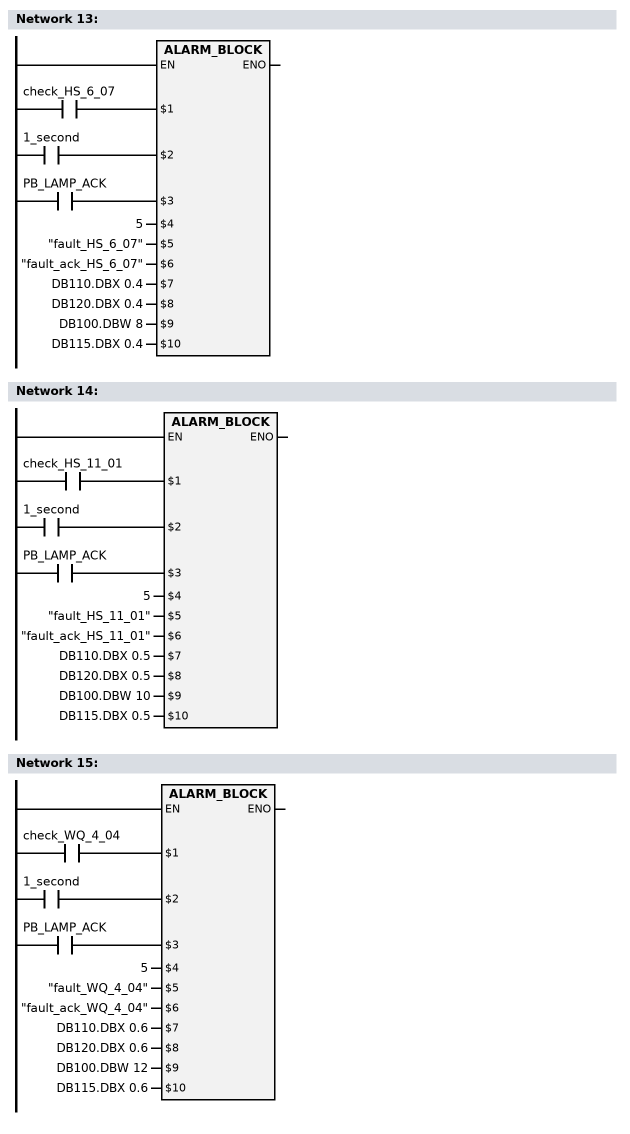
[picture p24: ALARM_HANDLING_STARCH networks 13-15]
NETWORK
TITLE =
      A     "check_HS_6_07";
      =     L 0.0;
      BLD   103;
      A     "1_second";
      =     L 0.1;
      BLD   103;
      A     "PB_LAMP_ACK";
      =     L 0.2;
      BLD   103;
      CALL  "ALARM_BLOCK" (
           $1                       := L 0.0,
           $2                       := L 0.1,
           $3                       := L 0.2,
           $4                       := 5,
           $5                       := "fault_HS_6_07",
           $6                       := "fault_ack_HS_6_07",
           $7                       := DB110.DBX 0.4,
           $8                       := DB120.DBX 0.4,
           $9                       := DB100.DBW 8,
           $10                      := DB115.DBX 0.4);
      NOP   0;
NETWORK
TITLE =
      A     "check_HS_11_01";
      =     L 0.0;
      BLD   103;
      A     "1_second";
      =     L 0.1;
      BLD   103;
      A     "PB_LAMP_ACK";
      =     L 0.2;
      BLD   103;
      CALL  "ALARM_BLOCK" (
           $1                       := L 0.0,
           $2                       := L 0.1,
           $3                       := L 0.2,
           $4                       := 5,
           $5                       := "fault_HS_11_01",
           $6                       := "fault_ack_HS_11_01",
           $7                       := DB110.DBX 0.5,
           $8                       := DB120.DBX 0.5,
           $9                       := DB100.DBW 10,
           $10                      := DB115.DBX 0.5);
      NOP   0;
NETWORK
TITLE =
      A     "check_WQ_4_04";
      =     L 0.0;
      BLD   103;
      A     "1_second";
      =     L 0.1;
      BLD   103;
      A     "PB_LAMP_ACK";
      =     L 0.2;
      BLD   103;
      CALL  "ALARM_BLOCK" (
           $1                       := L 0.0,
           $2                       := L 0.1,
           $3                       := L 0.2,
           $4                       := 5,
           $5                       := "fault_WQ_4_04",
           $6                       := "fault_ack_WQ_4_04",
           $7                       := DB110.DBX 0.6,
           $8                       := DB120.DBX 0.6,
           $9                       := DB100.DBW 12,
           $10                      := DB115.DBX 0.6);
      NOP   0;
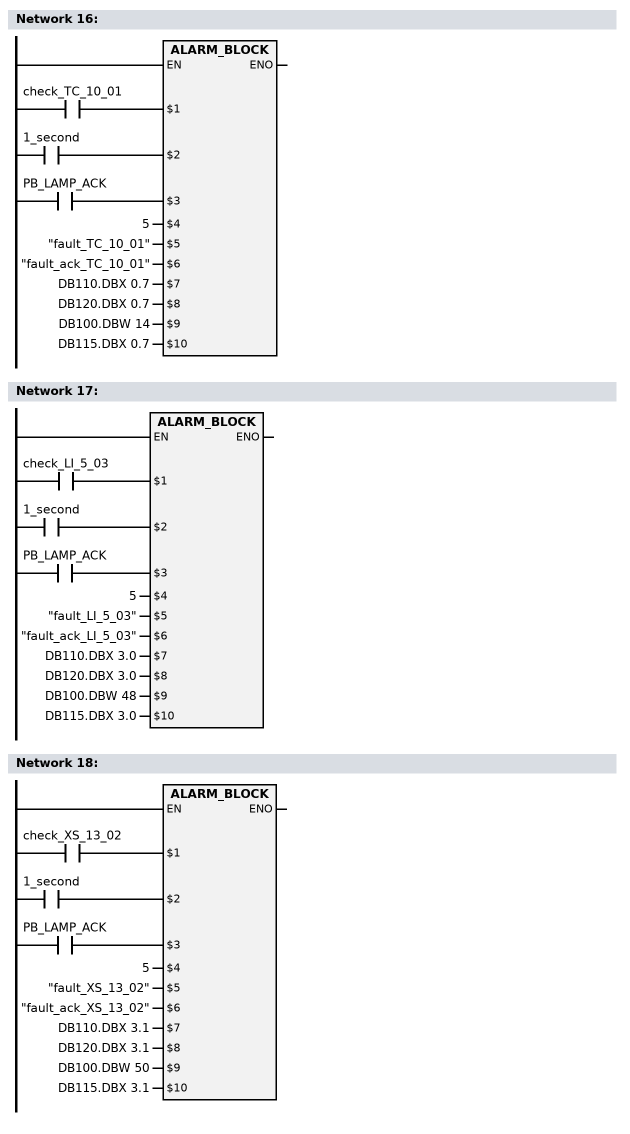
NETWORK
TITLE =
      A     "check_TC_10_01";
      =     L 0.0;
      BLD   103;
      A     "1_second";
      =     L 0.1;
      BLD   103;
      A     "PB_LAMP_ACK";
      =     L 0.2;
      BLD   103;
      CALL  "ALARM_BLOCK" (
           $1                       := L 0.0,
           $2                       := L 0.1,
           $3                       := L 0.2,
           $4                       := 5,
           $5                       := "fault_TC_10_01",
           $6                       := "fault_ack_TC_10_01",
           $7                       := DB110.DBX 0.7,
           $8                       := DB120.DBX 0.7,
           $9                       := DB100.DBW 14,
           $10                      := DB115.DBX 0.7);
      NOP   0;
NETWORK
TITLE =
      A     "check_LI_5_03";
      =     L 0.0;
      BLD   103;
      A     "1_second";
      =     L 0.1;
      BLD   103;
      A     "PB_LAMP_ACK";
      =     L 0.2;
      BLD   103;
      CALL  "ALARM_BLOCK" (
           $1                       := L 0.0,
           $2                       := L 0.1,
           $3                       := L 0.2,
           $4                       := 5,
           $5                       := "fault_LI_5_03",
           $6                       := "fault_ack_LI_5_03",
           $7                       := DB110.DBX 3.0,
           $8                       := DB120.DBX 3.0,
           $9                       := DB100.DBW 48,
           $10                      := DB115.DBX 3.0);
      NOP   0;
NETWORK
TITLE =
      A     "check_XS_13_02";
      =     L 0.0;
      BLD   103;
      A     "1_second";
      =     L 0.1;
      BLD   103;
      A     "PB_LAMP_ACK";
      =     L 0.2;
      BLD   103;
      CALL  "ALARM_BLOCK" (
           $1                       := L 0.0,
           $2                       := L 0.1,
           $3                       := L 0.2,
           $4                       := 5,
           $5                       := "fault_XS_13_02",
           $6                       := "fault_ack_XS_13_02",
           $7                       := DB110.DBX 3.1,
           $8                       := DB120.DBX 3.1,
           $9                       := DB100.DBW 50,
           $10                      := DB115.DBX 3.1);
      NOP   0;
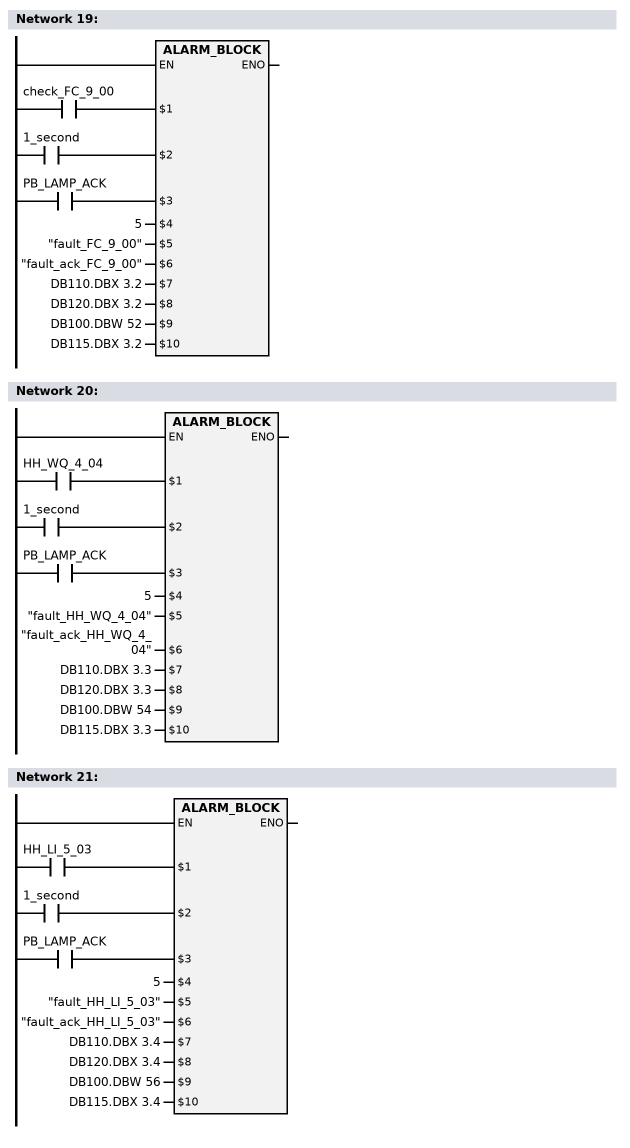
NETWORK
TITLE =
      A     "check_FC_9_00";
      =     L 0.0;
      BLD   103;
      A     "1_second";
      =     L 0.1;
      BLD   103;
      A     "PB_LAMP_ACK";
      =     L 0.2;
      BLD   103;
      CALL  "ALARM_BLOCK" (
           $1                       := L 0.0,
           $2                       := L 0.1,
           $3                       := L 0.2,
           $4                       := 5,
           $5                       := "fault_FC_9_00",
           $6                       := "fault_ack_FC_9_00",
           $7                       := DB110.DBX 3.2,
           $8                       := DB120.DBX 3.2,
           $9                       := DB100.DBW 52,
           $10                      := DB115.DBX 3.2);
      NOP   0;
NETWORK
TITLE =
      A     "HH_WQ_4_04";
      =     L 0.0;
      BLD   103;
      A     "1_second";
      =     L 0.1;
      BLD   103;
      A     "PB_LAMP_ACK";
      =     L 0.2;
      BLD   103;
      CALL  "ALARM_BLOCK" (
           $1                       := L 0.0,
           $2                       := L 0.1,
           $3                       := L 0.2,
           $4                       := 5,
           $5                       := "fault_HH_WQ_4_04",
           $6                       := "fault_ack_HH_WQ_4_04",
           $7                       := DB110.DBX 3.3,
           $8                       := DB120.DBX 3.3,
           $9                       := DB100.DBW 54,
           $10                      := DB115.DBX 3.3);
      NOP   0;
NETWORK
TITLE =
      A     "HH_LI_5_03";
      =     L 0.0;
      BLD   103;
      A     "1_second";
      =     L 0.1;
      BLD   103;
      A     "PB_LAMP_ACK";
      =     L 0.2;
      BLD   103;
      CALL  "ALARM_BLOCK" (
           $1                       := L 0.0,
           $2                       := L 0.1,
           $3                       := L 0.2,
           $4                       := 5,
           $5                       := "fault_HH_LI_5_03",
           $6                       := "fault_ack_HH_LI_5_03",
           $7                       := DB110.DBX 3.4,
           $8                       := DB120.DBX 3.4,
           $9                       := DB100.DBW 56,
           $10                      := DB115.DBX 3.4);
      NOP   0;
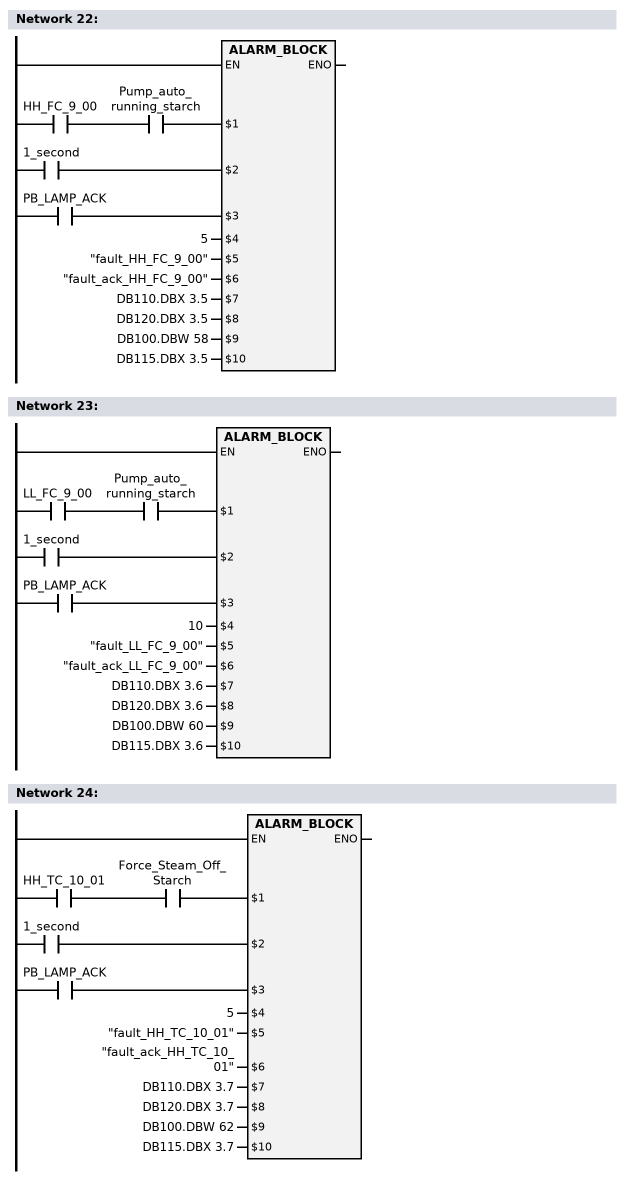
NETWORK
TITLE =
      A     "HH_FC_9_00";
      A     "Pump_auto_running_starch";
      =     L 0.0;
      BLD   103;
      A     "1_second";
      =     L 0.1;
      BLD   103;
      A     "PB_LAMP_ACK";
      =     L 0.2;
      BLD   103;
      CALL  "ALARM_BLOCK" (
           $1                       := L 0.0,
           $2                       := L 0.1,
           $3                       := L 0.2,
           $4                       := 5,
           $5                       := "fault_HH_FC_9_00",
           $6                       := "fault_ack_HH_FC_9_00",
           $7                       := DB110.DBX 3.5,
           $8                       := DB120.DBX 3.5,
           $9                       := DB100.DBW 58,
           $10                      := DB115.DBX 3.5);
      NOP   0;
NETWORK
TITLE =
      A     "LL_FC_9_00";
      A     "Pump_auto_running_starch";
      =     L 0.0;
      BLD   103;
      A     "1_second";
      =     L 0.1;
      BLD   103;
      A     "PB_LAMP_ACK";
      =     L 0.2;
      BLD   103;
      CALL  "ALARM_BLOCK" (
           $1                       := L 0.0,
           $2                       := L 0.1,
           $3                       := L 0.2,
           $4                       := 10,
           $5                       := "fault_LL_FC_9_00",
           $6                       := "fault_ack_LL_FC_9_00",
           $7                       := DB110.DBX 3.6,
           $8                       := DB120.DBX 3.6,
           $9                       := DB100.DBW 60,
           $10                      := DB115.DBX 3.6);
      NOP   0;
NETWORK
TITLE =
      A     "HH_TC_10_01";
      A     "Force_Steam_Off_Starch";
      =     L 0.0;
      BLD   103;
      A     "1_second";
      =     L 0.1;
      BLD   103;
      A     "PB_LAMP_ACK";
      =     L 0.2;
      BLD   103;
      CALL  "ALARM_BLOCK" (
           $1                       := L 0.0,
           $2                       := L 0.1,
           $3                       := L 0.2,
           $4                       := 5,
           $5                       := "fault_HH_TC_10_01",
           $6                       := "fault_ack_HH_TC_10_01",
           $7                       := DB110.DBX 3.7,
           $8                       := DB120.DBX 3.7,
           $9                       := DB100.DBW 62,
           $10                      := DB115.DBX 3.7);
      NOP   0;
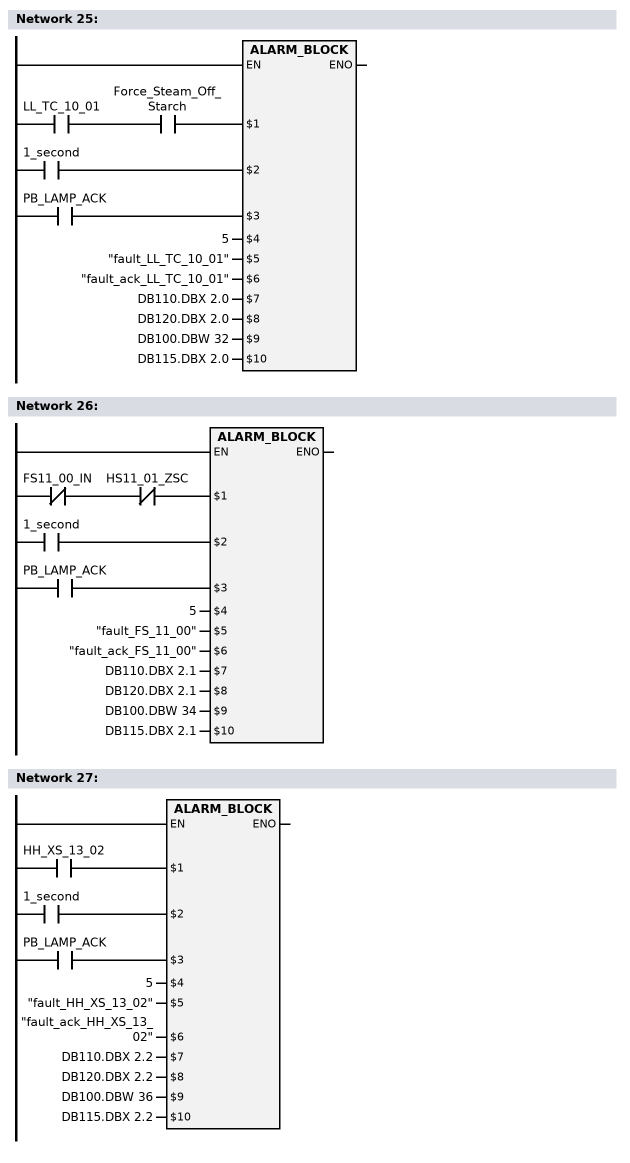
NETWORK
TITLE =
      A     "LL_TC_10_01";
      A     "Force_Steam_Off_Starch";
      =     L 0.0;
      BLD   103;
      A     "1_second";
      =     L 0.1;
      BLD   103;
      A     "PB_LAMP_ACK";
      =     L 0.2;
      BLD   103;
      CALL  "ALARM_BLOCK" (
           $1                       := L 0.0,
           $2                       := L 0.1,
           $3                       := L 0.2,
           $4                       := 5,
           $5                       := "fault_LL_TC_10_01",
           $6                       := "fault_ack_LL_TC_10_01",
           $7                       := DB110.DBX 2.0,
           $8                       := DB120.DBX 2.0,
           $9                       := DB100.DBW 32,
           $10                      := DB115.DBX 2.0);
      NOP   0;
NETWORK
TITLE =
      AN    "FS11_00_IN";
      AN    "HS11_01_ZSC";
      =     L 0.0;
      BLD   103;
      A     "1_second";
      =     L 0.1;
      BLD   103;
      A     "PB_LAMP_ACK";
      =     L 0.2;
      BLD   103;
      CALL  "ALARM_BLOCK" (
           $1                       := L 0.0,
           $2                       := L 0.1,
           $3                       := L 0.2,
           $4                       := 5,
           $5                       := "fault_FS_11_00",
           $6                       := "fault_ack_FS_11_00",
           $7                       := DB110.DBX 2.1,
           $8                       := DB120.DBX 2.1,
           $9                       := DB100.DBW 34,
           $10                      := DB115.DBX 2.1);
      NOP   0;
NETWORK
TITLE =
      A     "HH_XS_13_02";
      =     L 0.0;
      BLD   103;
      A     "1_second";
      =     L 0.1;
      BLD   103;
      A     "PB_LAMP_ACK";
      =     L 0.2;
      BLD   103;
      CALL  "ALARM_BLOCK" (
           $1                       := L 0.0,
           $2                       := L 0.1,
           $3                       := L 0.2,
           $4                       := 5,
           $5                       := "fault_HH_XS_13_02",
           $6                       := "fault_ack_HH_XS_13_02",
           $7                       := DB110.DBX 2.2,
           $8                       := DB120.DBX 2.2,
           $9                       := DB100.DBW 36,
           $10                      := DB115.DBX 2.2);
      NOP   0;
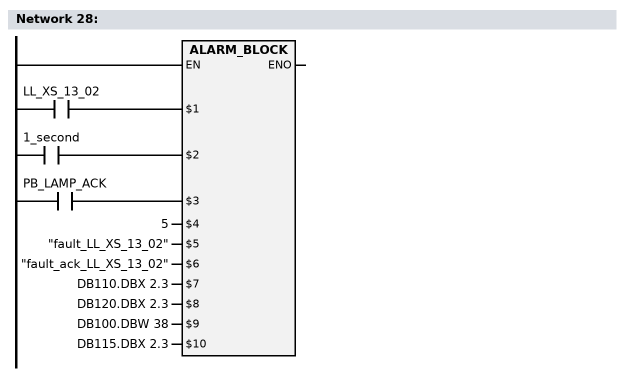
NETWORK
TITLE =
      A     "LL_XS_13_02";
      =     L 0.0;
      BLD   103;
      A     "1_second";
      =     L 0.1;
      BLD   103;
      A     "PB_LAMP_ACK";
      =     L 0.2;
      BLD   103;
      CALL  "ALARM_BLOCK" (
           $1                       := L 0.0,
           $2                       := L 0.1,
           $3                       := L 0.2,
           $4                       := 5,
           $5                       := "fault_LL_XS_13_02",
           $6                       := "fault_ack_LL_XS_13_02",
           $7                       := DB110.DBX 2.3,
           $8                       := DB120.DBX 2.3,
           $9                       := DB100.DBW 38,
           $10                      := DB115.DBX 2.3);
      NOP   0;
END_FUNCTION_BLOCK

FUNCTION_BLOCK "ALARM_HANDLING_CaCO3"	// FB 32
AUTHOR : GAW-LK
FAMILY : ALARM
NAME : ALARMS
VERSION : 0.1
BEGIN
// (block stored without names or comments; labels and parameter names are numbered)
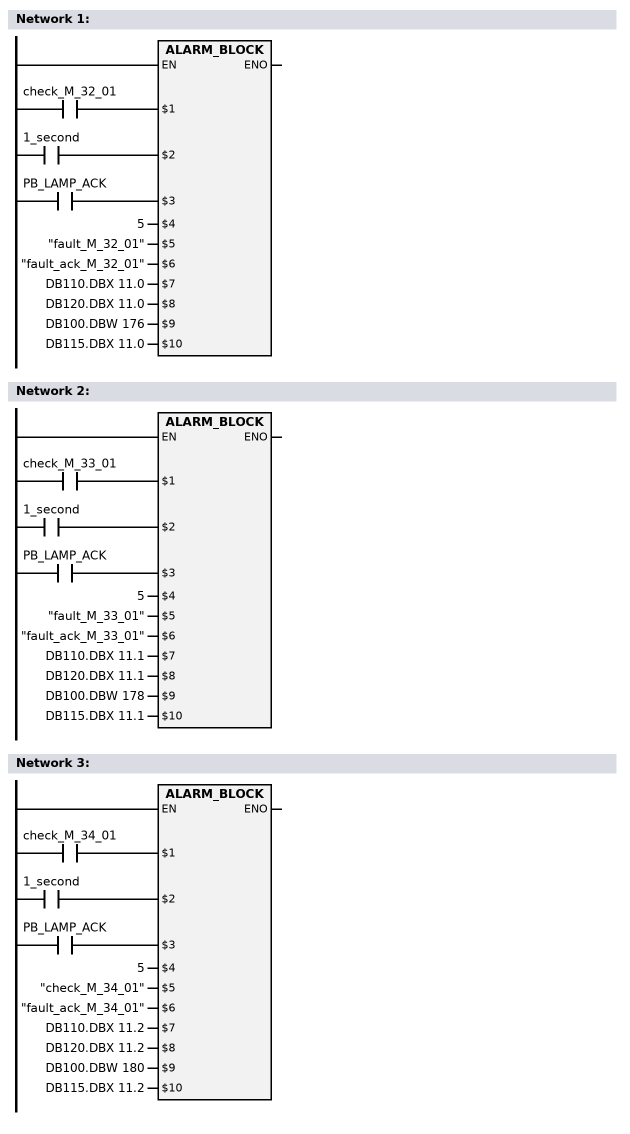
NETWORK
TITLE =
      A     "check_M_32_01";
      =     L 0.0;
      BLD   103;
      A     "1_second";
      =     L 0.1;
      BLD   103;
      A     "PB_LAMP_ACK";
      =     L 0.2;
      BLD   103;
      CALL  "ALARM_BLOCK" (
           $1                       := L 0.0,
           $2                       := L 0.1,
           $3                       := L 0.2,
           $4                       := 5,
           $5                       := "fault_M_32_01",
           $6                       := "fault_ack_M_32_01",
           $7                       := DB110.DBX 11.0,
           $8                       := DB120.DBX 11.0,
           $9                       := DB100.DBW 176,
           $10                      := DB115.DBX 11.0);
      NOP   0;
NETWORK
TITLE =
      A     "check_M_33_01";
      =     L 0.0;
      BLD   103;
      A     "1_second";
      =     L 0.1;
      BLD   103;
      A     "PB_LAMP_ACK";
      =     L 0.2;
      BLD   103;
      CALL  "ALARM_BLOCK" (
           $1                       := L 0.0,
           $2                       := L 0.1,
           $3                       := L 0.2,
           $4                       := 5,
           $5                       := "fault_M_33_01",
           $6                       := "fault_ack_M_33_01",
           $7                       := DB110.DBX 11.1,
           $8                       := DB120.DBX 11.1,
           $9                       := DB100.DBW 178,
           $10                      := DB115.DBX 11.1);
      NOP   0;
NETWORK
TITLE =
      A     "check_M_34_01";
      =     L 0.0;
      BLD   103;
      A     "1_second";
      =     L 0.1;
      BLD   103;
      A     "PB_LAMP_ACK";
      =     L 0.2;
      BLD   103;
      CALL  "ALARM_BLOCK" (
           $1                       := L 0.0,
           $2                       := L 0.1,
           $3                       := L 0.2,
           $4                       := 5,
           $5                       := "check_M_34_01",
           $6                       := "fault_ack_M_34_01",
           $7                       := DB110.DBX 11.2,
           $8                       := DB120.DBX 11.2,
           $9                       := DB100.DBW 180,
           $10                      := DB115.DBX 11.2);
      NOP   0;
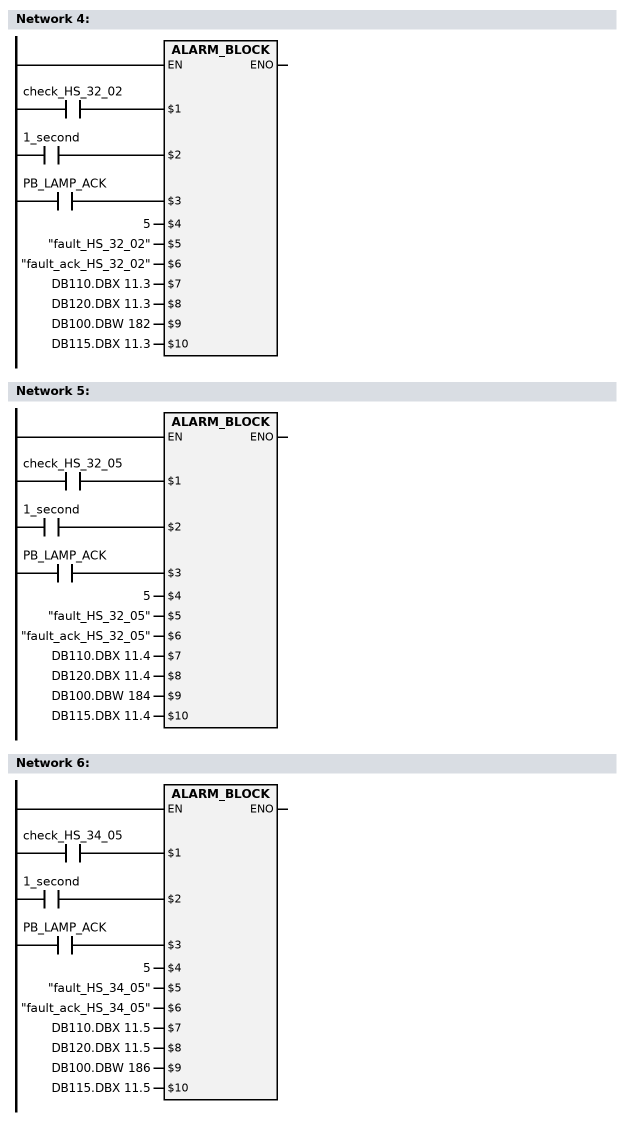
NETWORK
TITLE =
      A     "check_HS_32_02";
      =     L 0.0;
      BLD   103;
      A     "1_second";
      =     L 0.1;
      BLD   103;
      A     "PB_LAMP_ACK";
      =     L 0.2;
      BLD   103;
      CALL  "ALARM_BLOCK" (
           $1                       := L 0.0,
           $2                       := L 0.1,
           $3                       := L 0.2,
           $4                       := 5,
           $5                       := "fault_HS_32_02",
           $6                       := "fault_ack_HS_32_02",
           $7                       := DB110.DBX 11.3,
           $8                       := DB120.DBX 11.3,
           $9                       := DB100.DBW 182,
           $10                      := DB115.DBX 11.3);
      NOP   0;
NETWORK
TITLE =
      A     "check_HS_32_05";
      =     L 0.0;
      BLD   103;
      A     "1_second";
      =     L 0.1;
      BLD   103;
      A     "PB_LAMP_ACK";
      =     L 0.2;
      BLD   103;
      CALL  "ALARM_BLOCK" (
           $1                       := L 0.0,
           $2                       := L 0.1,
           $3                       := L 0.2,
           $4                       := 5,
           $5                       := "fault_HS_32_05",
           $6                       := "fault_ack_HS_32_05",
           $7                       := DB110.DBX 11.4,
           $8                       := DB120.DBX 11.4,
           $9                       := DB100.DBW 184,
           $10                      := DB115.DBX 11.4);
      NOP   0;
NETWORK
TITLE =
      A     "check_HS_34_05";
      =     L 0.0;
      BLD   103;
      A     "1_second";
      =     L 0.1;
      BLD   103;
      A     "PB_LAMP_ACK";
      =     L 0.2;
      BLD   103;
      CALL  "ALARM_BLOCK" (
           $1                       := L 0.0,
           $2                       := L 0.1,
           $3                       := L 0.2,
           $4                       := 5,
           $5                       := "fault_HS_34_05",
           $6                       := "fault_ack_HS_34_05",
           $7                       := DB110.DBX 11.5,
           $8                       := DB120.DBX 11.5,
           $9                       := DB100.DBW 186,
           $10                      := DB115.DBX 11.5);
      NOP   0;
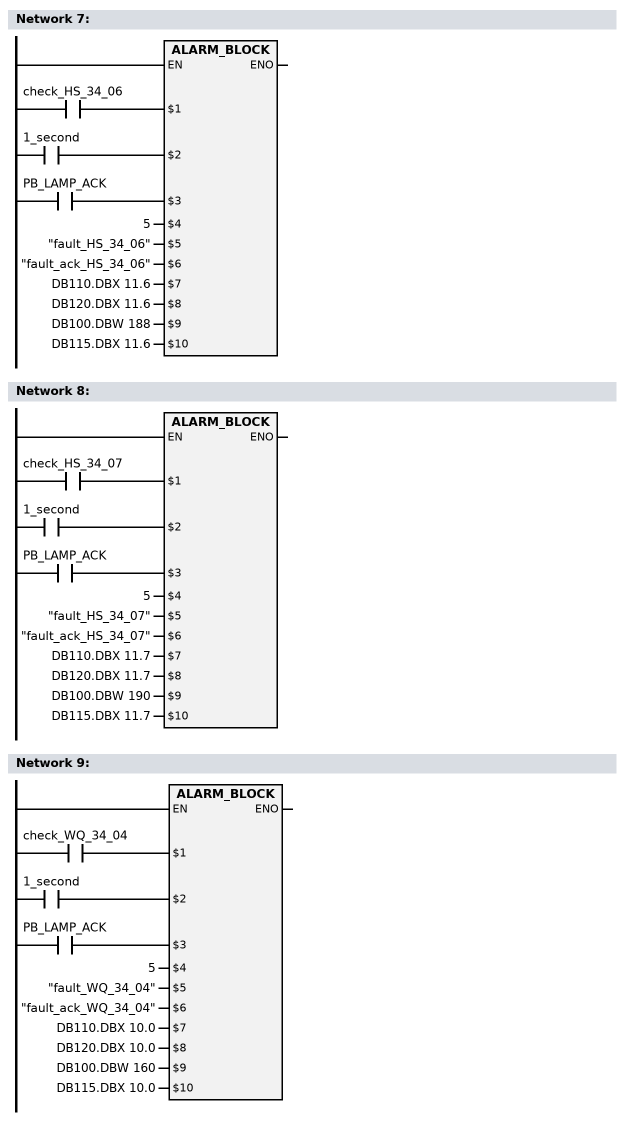
NETWORK
TITLE =
      A     "check_HS_34_06";
      =     L 0.0;
      BLD   103;
      A     "1_second";
      =     L 0.1;
      BLD   103;
      A     "PB_LAMP_ACK";
      =     L 0.2;
      BLD   103;
      CALL  "ALARM_BLOCK" (
           $1                       := L 0.0,
           $2                       := L 0.1,
           $3                       := L 0.2,
           $4                       := 5,
           $5                       := "fault_HS_34_06",
           $6                       := "fault_ack_HS_34_06",
           $7                       := DB110.DBX 11.6,
           $8                       := DB120.DBX 11.6,
           $9                       := DB100.DBW 188,
           $10                      := DB115.DBX 11.6);
      NOP   0;
NETWORK
TITLE =
      A     "check_HS_34_07";
      =     L 0.0;
      BLD   103;
      A     "1_second";
      =     L 0.1;
      BLD   103;
      A     "PB_LAMP_ACK";
      =     L 0.2;
      BLD   103;
      CALL  "ALARM_BLOCK" (
           $1                       := L 0.0,
           $2                       := L 0.1,
           $3                       := L 0.2,
           $4                       := 5,
           $5                       := "fault_HS_34_07",
           $6                       := "fault_ack_HS_34_07",
           $7                       := DB110.DBX 11.7,
           $8                       := DB120.DBX 11.7,
           $9                       := DB100.DBW 190,
           $10                      := DB115.DBX 11.7);
      NOP   0;
NETWORK
TITLE =
      A     "check_WQ_34_04";
      =     L 0.0;
      BLD   103;
      A     "1_second";
      =     L 0.1;
      BLD   103;
      A     "PB_LAMP_ACK";
      =     L 0.2;
      BLD   103;
      CALL  "ALARM_BLOCK" (
           $1                       := L 0.0,
           $2                       := L 0.1,
           $3                       := L 0.2,
           $4                       := 5,
           $5                       := "fault_WQ_34_04",
           $6                       := "fault_ack_WQ_34_04",
           $7                       := DB110.DBX 10.0,
           $8                       := DB120.DBX 10.0,
           $9                       := DB100.DBW 160,
           $10                      := DB115.DBX 10.0);
      NOP   0;
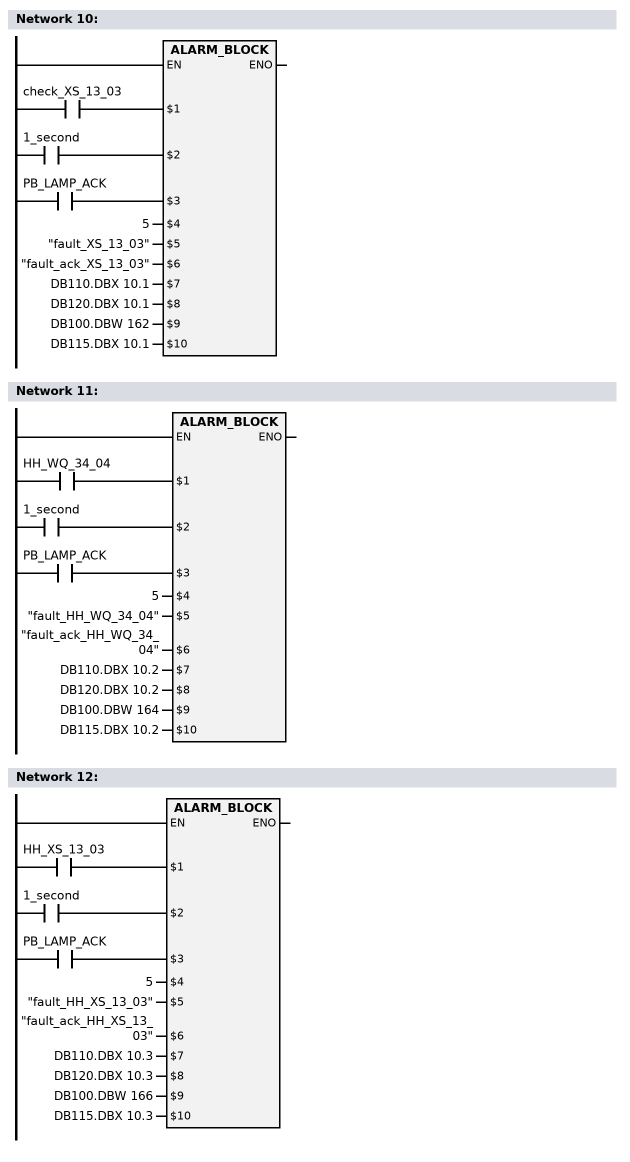
NETWORK
TITLE =
      A     "check_XS_13_03";
      =     L 0.0;
      BLD   103;
      A     "1_second";
      =     L 0.1;
      BLD   103;
      A     "PB_LAMP_ACK";
      =     L 0.2;
      BLD   103;
      CALL  "ALARM_BLOCK" (
           $1                       := L 0.0,
           $2                       := L 0.1,
           $3                       := L 0.2,
           $4                       := 5,
           $5                       := "fault_XS_13_03",
           $6                       := "fault_ack_XS_13_03",
           $7                       := DB110.DBX 10.1,
           $8                       := DB120.DBX 10.1,
           $9                       := DB100.DBW 162,
           $10                      := DB115.DBX 10.1);
      NOP   0;
NETWORK
TITLE =
      A     "HH_WQ_34_04";
      =     L 0.0;
      BLD   103;
      A     "1_second";
      =     L 0.1;
      BLD   103;
      A     "PB_LAMP_ACK";
      =     L 0.2;
      BLD   103;
      CALL  "ALARM_BLOCK" (
           $1                       := L 0.0,
           $2                       := L 0.1,
           $3                       := L 0.2,
           $4                       := 5,
           $5                       := "fault_HH_WQ_34_04",
           $6                       := "fault_ack_HH_WQ_34_04",
           $7                       := DB110.DBX 10.2,
           $8                       := DB120.DBX 10.2,
           $9                       := DB100.DBW 164,
           $10                      := DB115.DBX 10.2);
      NOP   0;
NETWORK
TITLE =
      A     "HH_XS_13_03";
      =     L 0.0;
      BLD   103;
      A     "1_second";
      =     L 0.1;
      BLD   103;
      A     "PB_LAMP_ACK";
      =     L 0.2;
      BLD   103;
      CALL  "ALARM_BLOCK" (
           $1                       := L 0.0,
           $2                       := L 0.1,
           $3                       := L 0.2,
           $4                       := 5,
           $5                       := "fault_HH_XS_13_03",
           $6                       := "fault_ack_HH_XS_13_03",
           $7                       := DB110.DBX 10.3,
           $8                       := DB120.DBX 10.3,
           $9                       := DB100.DBW 166,
           $10                      := DB115.DBX 10.3);
      NOP   0;
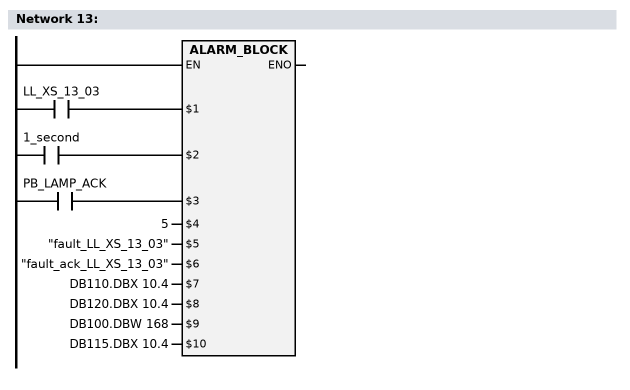
NETWORK
TITLE =
      A     "LL_XS_13_03";
      =     L 0.0;
      BLD   103;
      A     "1_second";
      =     L 0.1;
      BLD   103;
      A     "PB_LAMP_ACK";
      =     L 0.2;
      BLD   103;
      CALL  "ALARM_BLOCK" (
           $1                       := L 0.0,
           $2                       := L 0.1,
           $3                       := L 0.2,
           $4                       := 5,
           $5                       := "fault_LL_XS_13_03",
           $6                       := "fault_ack_LL_XS_13_03",
           $7                       := DB110.DBX 10.4,
           $8                       := DB120.DBX 10.4,
           $9                       := DB100.DBW 168,
           $10                      := DB115.DBX 10.4);
      NOP   0;
END_FUNCTION_BLOCK

FUNCTION_BLOCK "ALARM"	// FB 33
AUTHOR : GAW-LK
FAMILY : ALARM
NAME : ALARM
VERSION : 0.1
BEGIN
// (block stored without names or comments; labels and parameter names are numbered)
NETWORK
TITLE =
      L     DB110.DBW 0;
      L     0;
      ==I;
      =     L 1.0;
      L     DB110.DBW 2;
      L     0;
      ==I;
      =     L 1.1;
      L     DB110.DBW 4;
      L     0;
      ==I;
      =     L 1.2;
      L     DB110.DBW 6;
      L     0;
      ==I;
      =     L 1.3;
      L     DB110.DBW 8;
      L     0;
      ==I;
      =     L 1.4;
      L     DB110.DBW 10;
      L     0;
      ==I;
      =     L 1.5;
      L     DB110.DBW 12;
      L     0;
      ==I;
      =     L 1.6;
      L     DB110.DBW 14;
      L     0;
      ==I;
      =     L 1.7;
      L     DB110.DBW 16;
      L     0;
      ==I;
      =     L 2.0;
      ON    L 1.0;
      ON    L 1.1;
      ON    L 1.2;
      ON    L 1.3;
      ON    L 1.4;
      L     S5T#500MS;
      SD    T 5;
      A     T 5;
      =     L 100.0;
      ON    L 1.5;
      ON    L 1.6;
      ON    L 1.7;
      ON    L 2.0;
      L     S5T#500MS;
      SD    T 6;
      A     T 6;
      =     L 100.1;
NETWORK
TITLE =
      L     DB110.DBW 0;
      L     DB120.DBW 0;
      ==I;
      =     L 4.0;
      L     DB110.DBW 2;
      L     DB120.DBW 2;
      ==I;
      =     L 4.1;
      L     DB110.DBW 4;
      L     DB120.DBW 4;
      ==I;
      =     L 4.2;
      L     DB110.DBW 6;
      L     DB120.DBW 6;
      ==I;
      =     L 4.3;
      L     DB110.DBW 8;
      L     DB120.DBW 8;
      ==I;
      =     L 4.4;
      L     DB110.DBW 10;
      L     DB120.DBW 10;
      ==I;
      =     L 4.5;
      L     DB110.DBW 12;
      L     DB120.DBW 12;
      ==I;
      =     L 4.6;
      L     DB110.DBW 14;
      L     DB120.DBW 14;
      ==I;
      =     L 4.7;
      L     DB110.DBW 16;
      L     DB120.DBW 16;
      ==I;
      =     L 5.0;
      ON    L 4.0;
      ON    L 4.1;
      ON    L 4.2;
      ON    L 4.3;
      ON    L 4.4;
      ON    L 4.5;
      ON    L 4.6;
      ON    L 4.7;
      ON    L 5.0;
      L     S5T#500MS;
      SD    T 7;
      A     T 7;
      =     "XA13_01_ON";
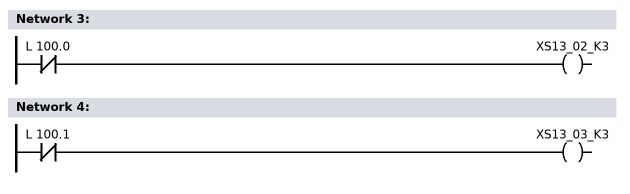
NETWORK
TITLE =
      AN    L 100.0;
      =     "XS13_02_K3";
NETWORK
TITLE =
      AN    L 100.1;
      =     "XS13_03_K3";
END_FUNCTION_BLOCK

// FB 41: know-how protected block, not included

FUNCTION_BLOCK "Batch"	// FB 90
VERSION : 0.1
BEGIN
// (block stored without names or comments; labels and parameter names are numbered)
NETWORK
TITLE =
      TAR1  LD 4;
NETWORK
TITLE =
      A     DIX [AR2,P#0.0];
      AN    DIX [AR2,P#16.0];
      =     DIX [AR2,P#398.1];
      =     DIX [AR2,P#16.1];
      S     DIX [AR2,P#16.0];
      A     DIX [AR2,P#14.1];
      S     DIX [AR2,P#394.0];
      A     DIX [AR2,P#394.0];
      R     DIX [AR2,P#16.0];
      L     DIW [AR2,P#400.0];
      T     DIW [AR2,P#18.0];
      O     DIX [AR2,P#398.1];
      O     DIX [AR2,P#394.0];
      JC    M023;
      A     DIX [AR2,P#16.0];
      JC    M001;
      BEU;
M001: NOP   0;
      SET;
      R     L 22.0;
      AN    DIX [AR2,P#398.0];
      JC    M002;
      R     DIX [AR2,P#398.0];
      L     DIW [AR2,P#396.0];
      L     1;
      +I;
      T     DIW [AR2,P#396.0];
      L     DIW [AR2,P#10.0];
      >=I;
      =     DIX [AR2,P#394.0];
      JC    M027;
M002: NOP   0;
      LAR1  P#DIX 20.0;
      L     0;
      T     LW 8;
M003: L     DIW [AR2,P#396.0];
      L     LW 8;
      ==I;
      JC    M004;
      L     DIW [AR2,P#396.0];
      L     272;
      *I;
      +AR1;
      L     LW 8;
      L     1;
      +I;
      T     LW 8;
      TAR1  LD 16;
      LOOP  M003;
M004: NOP   0;
      SET;
      R      [AR1,P#32.2];
      L     0;
      L     W [AR1,P#20.0];
      ==I;
      JC    M008;
      L     1;
      L     W [AR1,P#20.0];
      ==I;
      JC    M009;
      L     2;
      L     W [AR1,P#20.0];
      ==I;
      JC    M005;
      L     3;
      L     W [AR1,P#20.0];
      ==I;
      JC    M006;
      JU    M007;
M005: S      [AR1,P#32.0];
      SET;
      =      [AR1,P#32.3];
      A      [AR1,P#32.3];
      A      [AR1,P#32.4];
      JC    M016;
      JU    M018;
M006: A      [AR1,P#32.0];
      JC    M015;
      L     L#0;
      T     DID [AR2,P#402.0];
      SET;
      S      [AR1,P#32.0];
      JU    M015;
M007: NOP   0;
M008: L     DID [AR2,P#2.0];
      JU    M013;
M009: SET;
      =     L 22.0;
      L     W [AR1,P#30.0];
      L     1;
      -I;
      L     DIW [AR2,P#396.0];
      -I;
      T     LW 20;
      L     0;
      >I;
      JC    M010;
      JU    M012;
M010: LAR1  LD 16;
      L     LW 20;
      L     272;
      *I;
      +AR1;
      L     DID [AR2,P#2.0];
      T     D [AR1,P#16.0];
      A      [AR1,P#32.0];
      JC    M011;
      L     D [AR1,P#16.0];
      T     D [AR1,P#12.0];
      L     0.000000e+00;
      T     D [AR1,P#4.0];
      SET;
      S      [AR1,P#32.2];
      S      [AR1,P#32.0];
M011: L     D [AR1,P#16.0];
      L     D [AR1,P#12.0];
      -R;
      L     D [AR1,P#4.0];
      +R;
      T     D [AR1,P#4.0];
      L     D [AR1,P#16.0];
      T     D [AR1,P#12.0];
      LAR1  LD 16;
M012: L     DID [AR2,P#6.0];
      JU    M013;
M013: T     D [AR1,P#16.0];
      A      [AR1,P#32.0];
      JC    M014;
      L     0.000000e+00;
      T     D [AR1,P#4.0];
      T     D [AR1,P#12.0];
      L     L#0;
      T     DID [AR2,P#402.0];
      A     L 22.0;
      JC    M014;
      L     D [AR1,P#16.0];
      T     D [AR1,P#12.0];
M014: L     D [AR1,P#16.0];
      L     D [AR1,P#12.0];
      -R;
      L     D [AR1,P#4.0];
      +R;
      T     D [AR1,P#4.0];
      L     D [AR1,P#16.0];
      T     D [AR1,P#12.0];
      L     D [AR1,P#0.0];
      L     D [AR1,P#8.0];
      -R;
      L     D [AR1,P#4.0];
      >R;
      =     L 10.0;
      SET;
      S      [AR1,P#32.0];
      A     L 10.0;
      AN     [AR1,P#32.2];
      =      [AR1,P#32.1];
      A     L 10.0;
      JC    M017;
M015: L     3;
      L     W [AR1,P#20.0];
      ==I;
      A     DIX [AR2,P#14.0];
      JC    M018;
      L     DIW [AR2,P#12.0];
      L     DID [AR2,P#402.0];
      +D;
      T     DID [AR2,P#402.0];
      L     1000;
      /D;
      T     D [AR1,P#26.0];
      L     D [AR1,P#22.0];
      >=D;
M016: S     DIX [AR2,P#398.0];
      R      [AR1,P#32.0];
      JU    M018;
M017: L     0;
      T     DID [AR2,P#402.0];
M018: NOP   0;
      L     0;
      T     LW 24;
      T     DIW [AR2,P#400.0];
M019: LAR1  P#DIX 20.0;
      L     LW 24;
      L     272;
      *I;
      +AR1;
      AN     [AR1,P#32.0];
      JC    M020;
      L     LW 24;
      L     1;
      SLW;
      L     DIW [AR2,P#400.0];
      +I;
      T     DIW [AR2,P#400.0];
      JU    M021;
M020: L     LW 24;
      L     0;
      SLW;
      L     DIW [AR2,P#400.0];
      +I;
      T     DIW [AR2,P#400.0];
M021: L     1;
      L     LW 24;
      +I;
      T     LW 24;
      L     DIW [AR2,P#10.0];
      >=I;
      JC    M022;
      LOOP  M019;
M022: JU    M027;
M023: L     0;
      T     LW 24;
      T     DIW [AR2,P#400.0];
M024: LAR1  P#DIX 20.0;
      L     LW 24;
      L     272;
      *I;
      +AR1;
      A     DIX [AR2,P#394.0];
      JC    M025;
      L     0.000000e+00;
      T     D [AR1,P#16.0];
      T     D [AR1,P#12.0];
      T     D [AR1,P#4.0];
      L     L#0;
      T     D [AR1,P#26.0];
      L     0;
      T     W [AR1,P#26.0];
M025: SET;
      R      [AR1,P#32.0];
      R      [AR1,P#32.2];
      R      [AR1,P#32.1];
      R      [AR1,P#32.3];
      R      [AR1,P#32.4];
      L     1;
      L     LW 24;
      +I;
      T     LW 24;
      L     DIW [AR2,P#10.0];
      >=I;
      JC    M026;
      LOOP  M024;
M026: A     DIX [AR2,P#394.0];
      R     DIX [AR2,P#394.0];
      L     0;
      T     DIW [AR2,P#396.0];
      T     DIW [AR2,P#400.0];
NETWORK
TITLE =
M027: LAR1  LD 4;
END_FUNCTION_BLOCK

FUNCTION_BLOCK "Control"	// FB 110
AUTHOR : gaw-be
FAMILY : PID
NAME : Control
VERSION : 0.1
BEGIN
// (block stored without names or comments; labels and parameter names are numbered)
NETWORK
TITLE =
      L     DID [AR2,P#24.0];
      L     T#10MS;
      <D;
      JC    M001;
      L     DID [AR2,P#24.0];
      L     T#1S;
      >D;
      JC    M001;
      JU    M002;
M001: T     DID [AR2,P#24.0];
M002: NOP   0;
      BLD   18;
      T     LD 22;
      TAK;
      T     LD 26;
      L     DIW [AR2,P#34.0];
      T     LW 30;
      OPN   DB [LW 30];
      L     DID [AR2,P#36.0];
      LAR1;
      L     LD 26;
      L     LD 22;
      L     D [AR1,P#36.0];
      L     T#10MS;
      <D;
      JC    M003;
      BLD   18;
      T     LD 22;
      TAK;
      T     LD 26;
      L     DIW [AR2,P#34.0];
      T     LW 30;
      OPN   DB [LW 30];
      L     DID [AR2,P#36.0];
      LAR1;
      L     LD 26;
      L     LD 22;
      L     D [AR1,P#36.0];
      L     T#1M;
      >D;
      JC    M003;
      JU    M004;
M003: BLD   18;
      T     LD 22;
      TAK;
      T     LD 26;
      L     DIW [AR2,P#34.0];
      T     LW 30;
      OPN   DB [LW 30];
      L     DID [AR2,P#36.0];
      LAR1;
      L     LD 26;
      L     LD 22;
      T     D [AR1,P#36.0];
M004: NOP   0;
      BLD   18;
      T     LD 22;
      TAK;
      T     LD 26;
      L     DIW [AR2,P#34.0];
      T     LW 30;
      OPN   DB [LW 30];
      L     DID [AR2,P#36.0];
      LAR1;
      L     LD 26;
      L     LD 22;
      L     D [AR1,P#40.0];
      L     T#10MS;
      <D;
      JC    M005;
      BLD   18;
      T     LD 22;
      TAK;
      T     LD 26;
      L     DIW [AR2,P#34.0];
      T     LW 30;
      OPN   DB [LW 30];
      L     DID [AR2,P#36.0];
      LAR1;
      L     LD 26;
      L     LD 22;
      L     D [AR1,P#40.0];
      L     T#1M;
      >D;
      JC    M005;
      JU    M006;
M005: BLD   18;
      T     LD 22;
      TAK;
      T     LD 26;
      L     DIW [AR2,P#34.0];
      T     LW 30;
      OPN   DB [LW 30];
      L     DID [AR2,P#36.0];
      LAR1;
      L     LD 26;
      L     LD 22;
      T     D [AR1,P#40.0];
M006: NOP   0;
NETWORK
TITLE =
      BLD   18;
      T     LD 22;
      TAK;
      T     LD 26;
      L     DIW [AR2,P#34.0];
      T     LW 30;
      OPN   DB [LW 30];
      L     DID [AR2,P#36.0];
      LAR1;
      L     LD 26;
      L     LD 22;
      AN     [AR1,P#62.0];
      JC    M007;
      L     DID [AR2,P#24.0];
      DTR;
      BLD   18;
      T     LD 22;
      TAK;
      T     LD 26;
      L     DIW [AR2,P#34.0];
      T     LW 30;
      OPN   DB [LW 30];
      L     DID [AR2,P#36.0];
      LAR1;
      L     LD 26;
      L     LD 22;
      L     D [AR1,P#36.0];
      DTR;
      /R;
      T     LD 12;
      L     DID [AR2,P#0.0];
      BLD   18;
      T     LD 22;
      TAK;
      T     LD 26;
      L     DIW [AR2,P#34.0];
      T     LW 30;
      OPN   DB [LW 30];
      L     DID [AR2,P#36.0];
      LAR1;
      L     LD 26;
      L     LD 22;
      L     D [AR1,P#0.0];
      -R;
      L     LD 12;
      *R;
      BLD   18;
      T     LD 22;
      TAK;
      T     LD 26;
      L     DIW [AR2,P#34.0];
      T     LW 30;
      OPN   DB [LW 30];
      L     DID [AR2,P#36.0];
      LAR1;
      L     LD 26;
      L     LD 22;
      L     D [AR1,P#0.0];
      +R;
      BLD   18;
      T     LD 22;
      TAK;
      T     LD 26;
      L     DIW [AR2,P#34.0];
      T     LW 30;
      OPN   DB [LW 30];
      L     DID [AR2,P#36.0];
      LAR1;
      L     LD 26;
      L     LD 22;
      T     D [AR1,P#0.0];
      JU    M008;
M007: L     DID [AR2,P#0.0];
      BLD   18;
      T     LD 22;
      TAK;
      T     LD 26;
      L     DIW [AR2,P#34.0];
      T     LW 30;
      OPN   DB [LW 30];
      L     DID [AR2,P#36.0];
      LAR1;
      L     LD 26;
      L     LD 22;
      T     D [AR1,P#0.0];
M008: NOP   0;
      BLD   18;
      T     LD 22;
      TAK;
      T     LD 26;
      L     DIW [AR2,P#34.0];
      T     LW 30;
      OPN   DB [LW 30];
      L     DID [AR2,P#36.0];
      LAR1;
      L     LD 26;
      L     LD 22;
      AN     [AR1,P#62.1];
      JC    M009;
      L     DID [AR2,P#24.0];
      DTR;
      BLD   18;
      T     LD 22;
      TAK;
      T     LD 26;
      L     DIW [AR2,P#34.0];
      T     LW 30;
      OPN   DB [LW 30];
      L     DID [AR2,P#36.0];
      LAR1;
      L     LD 26;
      L     LD 22;
      L     D [AR1,P#40.0];
      DTR;
      /R;
      T     LD 12;
      L     DID [AR2,P#6.0];
      BLD   18;
      T     LD 22;
      TAK;
      T     LD 26;
      L     DIW [AR2,P#34.0];
      T     LW 30;
      OPN   DB [LW 30];
      L     DID [AR2,P#36.0];
      LAR1;
      L     LD 26;
      L     LD 22;
      L     D [AR1,P#4.0];
      -R;
      L     LD 12;
      *R;
      BLD   18;
      T     LD 22;
      TAK;
      T     LD 26;
      L     DIW [AR2,P#34.0];
      T     LW 30;
      OPN   DB [LW 30];
      L     DID [AR2,P#36.0];
      LAR1;
      L     LD 26;
      L     LD 22;
      L     D [AR1,P#4.0];
      +R;
      BLD   18;
      T     LD 22;
      TAK;
      T     LD 26;
      L     DIW [AR2,P#34.0];
      T     LW 30;
      OPN   DB [LW 30];
      L     DID [AR2,P#36.0];
      LAR1;
      L     LD 26;
      L     LD 22;
      T     D [AR1,P#4.0];
      JU    M010;
M009: L     DID [AR2,P#6.0];
      BLD   18;
      T     LD 22;
      TAK;
      T     LD 26;
      L     DIW [AR2,P#34.0];
      T     LW 30;
      OPN   DB [LW 30];
      L     DID [AR2,P#36.0];
      LAR1;
      L     LD 26;
      L     LD 22;
      T     D [AR1,P#4.0];
M010: NOP   0;
NETWORK
TITLE =
      L     DIB [AR2,P#4.0];
      BLD   18;
      T     LD 22;
      TAK;
      T     LD 26;
      L     DIW [AR2,P#34.0];
      T     LW 30;
      OPN   DB [LW 30];
      L     DID [AR2,P#36.0];
      LAR1;
      L     LD 26;
      L     LD 22;
      T     B [AR1,P#60.0];
      A     DIX [AR2,P#10.0];
      BLD   18;
      T     LD 22;
      TAK;
      T     LD 26;
      L     DIW [AR2,P#34.0];
      T     LW 30;
      OPN   DB [LW 30];
      L     DID [AR2,P#36.0];
      LAR1;
      L     LD 26;
      L     LD 22;
      =      [AR1,P#61.2];
      L     DID [AR2,P#12.0];
      BLD   18;
      T     LD 22;
      TAK;
      T     LD 26;
      L     DIW [AR2,P#34.0];
      T     LW 30;
      OPN   DB [LW 30];
      L     DID [AR2,P#36.0];
      LAR1;
      L     LD 26;
      L     LD 22;
      T     D [AR1,P#52.0];
      A     DIX [AR2,P#16.0];
      BLD   18;
      T     LD 22;
      TAK;
      T     LD 26;
      L     DIW [AR2,P#34.0];
      T     LW 30;
      OPN   DB [LW 30];
      L     DID [AR2,P#36.0];
      LAR1;
      L     LD 26;
      L     LD 22;
      =      [AR1,P#61.3];
      L     DID [AR2,P#18.0];
      BLD   18;
      T     LD 22;
      TAK;
      T     LD 26;
      L     DIW [AR2,P#34.0];
      T     LW 30;
      OPN   DB [LW 30];
      L     DID [AR2,P#36.0];
      LAR1;
      L     LD 26;
      L     LD 22;
      T     D [AR1,P#56.0];
      A     DIX [AR2,P#32.0];
      BLD   18;
      T     LD 22;
      TAK;
      T     LD 26;
      L     DIW [AR2,P#34.0];
      T     LW 30;
      OPN   DB [LW 30];
      L     DID [AR2,P#36.0];
      LAR1;
      L     LD 26;
      L     LD 22;
      =      [AR1,P#61.1];
      A     DIX [AR2,P#32.1];
      BLD   18;
      T     LD 22;
      TAK;
      T     LD 26;
      L     DIW [AR2,P#34.0];
      T     LW 30;
      OPN   DB [LW 30];
      L     DID [AR2,P#36.0];
      LAR1;
      L     LD 26;
      L     LD 22;
      =      [AR1,P#61.0];
      SET;
      =     L 6.1;
      R     L 6.0;
NETWORK
TITLE =
      BLD   18;
      T     LD 22;
      TAK;
      T     LD 26;
      L     DIW [AR2,P#40.0];
      T     LW 30;
      OPN   DB [LW 30];
      L     DID [AR2,P#42.0];
      LAR1;
      L     LD 26;
      L     LD 22;
      L     W [AR1,P#60.0];
      L     -1;
      ==I;
      BLD   18;
      T     LD 22;
      TAK;
      T     LD 26;
      L     DIW [AR2,P#40.0];
      T     LW 30;
      OPN   DB [LW 30];
      L     DID [AR2,P#42.0];
      LAR1;
      L     LD 26;
      L     LD 22;
      R      [AR1,P#62.0];
      L     DIW [AR2,P#22.0];
      BLD   18;
      T     LD 22;
      TAK;
      T     LD 26;
      L     DIW [AR2,P#40.0];
      T     LW 30;
      OPN   DB [LW 30];
      L     DID [AR2,P#42.0];
      LAR1;
      L     LD 26;
      L     LD 22;
      L     W [AR1,P#60.0];
      <>I;
      JC    M034;
      BLD   18;
      T     LD 22;
      TAK;
      T     LD 26;
      L     DIW [AR2,P#40.0];
      T     LW 30;
      OPN   DB [LW 30];
      L     DID [AR2,P#42.0];
      LAR1;
      L     LD 26;
      L     LD 22;
      A      [AR1,P#62.0];
      JC    M011;
      BLD   18;
      T     LD 22;
      TAK;
      T     LD 26;
      L     DIW [AR2,P#34.0];
      T     LW 30;
      OPN   DB [LW 30];
      L     DID [AR2,P#36.0];
      LAR1;
      L     LD 26;
      L     LD 22;
      L     D [AR1,P#8.0];
      BLD   18;
      T     LD 22;
      TAK;
      T     LD 26;
      L     DIW [AR2,P#40.0];
      T     LW 30;
      OPN   DB [LW 30];
      L     DID [AR2,P#42.0];
      LAR1;
      L     LD 26;
      L     LD 22;
      T     D [AR1,P#8.0];
      BLD   18;
      T     LD 22;
      TAK;
      T     LD 26;
      L     DIW [AR2,P#34.0];
      T     LW 30;
      OPN   DB [LW 30];
      L     DID [AR2,P#36.0];
      LAR1;
      L     LD 26;
      L     LD 22;
      L     D [AR1,P#16.0];
      BLD   18;
      T     LD 22;
      TAK;
      T     LD 26;
      L     DIW [AR2,P#40.0];
      T     LW 30;
      OPN   DB [LW 30];
      L     DID [AR2,P#42.0];
      LAR1;
      L     LD 26;
      L     LD 22;
      T     D [AR1,P#12.0];
      BLD   18;
      T     LD 22;
      TAK;
      T     LD 26;
      L     DIW [AR2,P#34.0];
      T     LW 30;
      OPN   DB [LW 30];
      L     DID [AR2,P#36.0];
      LAR1;
      L     LD 26;
      L     LD 22;
      A      [AR1,P#61.0];
      BLD   18;
      T     LD 22;
      TAK;
      T     LD 26;
      L     DIW [AR2,P#40.0];
      T     LW 30;
      OPN   DB [LW 30];
      L     DID [AR2,P#42.0];
      LAR1;
      L     LD 26;
      L     LD 22;
      =      [AR1,P#57.0];
      BLD   18;
      T     LD 22;
      TAK;
      T     LD 26;
      L     DIW [AR2,P#34.0];
      T     LW 30;
      OPN   DB [LW 30];
      L     DID [AR2,P#36.0];
      LAR1;
      L     LD 26;
      L     LD 22;
      A      [AR1,P#61.1];
      BLD   18;
      T     LD 22;
      TAK;
      T     LD 26;
      L     DIW [AR2,P#40.0];
      T     LW 30;
      OPN   DB [LW 30];
      L     DID [AR2,P#42.0];
      LAR1;
      L     LD 26;
      L     LD 22;
      =      [AR1,P#57.1];
      BLD   18;
      T     LD 22;
      TAK;
      T     LD 26;
      L     DIW [AR2,P#34.0];
      T     LW 30;
      OPN   DB [LW 30];
      L     DID [AR2,P#36.0];
      LAR1;
      L     LD 26;
      L     LD 22;
      L     D [AR1,P#20.0];
      BLD   18;
      T     LD 22;
      TAK;
      T     LD 26;
      L     DIW [AR2,P#40.0];
      T     LW 30;
      OPN   DB [LW 30];
      L     DID [AR2,P#42.0];
      LAR1;
      L     LD 26;
      L     LD 22;
      T     D [AR1,P#16.0];
      BLD   18;
      T     LD 22;
      TAK;
      T     LD 26;
      L     DIW [AR2,P#34.0];
      T     LW 30;
      OPN   DB [LW 30];
      L     DID [AR2,P#36.0];
      LAR1;
      L     LD 26;
      L     LD 22;
      A      [AR1,P#61.4];
      BLD   18;
      T     LD 22;
      TAK;
      T     LD 26;
      L     DIW [AR2,P#40.0];
      T     LW 30;
      OPN   DB [LW 30];
      L     DID [AR2,P#42.0];
      LAR1;
      L     LD 26;
      L     LD 22;
      =      [AR1,P#57.4];
      BLD   18;
      T     LD 22;
      TAK;
      T     LD 26;
      L     DIW [AR2,P#34.0];
      T     LW 30;
      OPN   DB [LW 30];
      L     DID [AR2,P#36.0];
      LAR1;
      L     LD 26;
      L     LD 22;
      A      [AR1,P#61.5];
      BLD   18;
      T     LD 22;
      TAK;
      T     LD 26;
      L     DIW [AR2,P#40.0];
      T     LW 30;
      OPN   DB [LW 30];
      L     DID [AR2,P#42.0];
      LAR1;
      L     LD 26;
      L     LD 22;
      =      [AR1,P#57.5];
      BLD   18;
      T     LD 22;
      TAK;
      T     LD 26;
      L     DIW [AR2,P#34.0];
      T     LW 30;
      OPN   DB [LW 30];
      L     DID [AR2,P#36.0];
      LAR1;
      L     LD 26;
      L     LD 22;
      L     D [AR1,P#24.0];
      L     1000;
      /D;
      BLD   18;
      T     LD 22;
      TAK;
      T     LD 26;
      L     DIW [AR2,P#40.0];
      T     LW 30;
      OPN   DB [LW 30];
      L     DID [AR2,P#42.0];
      LAR1;
      L     LD 26;
      L     LD 22;
      T     D [AR1,P#20.0];
      BLD   18;
      T     LD 22;
      TAK;
      T     LD 26;
      L     DIW [AR2,P#34.0];
      T     LW 30;
      OPN   DB [LW 30];
      L     DID [AR2,P#36.0];
      LAR1;
      L     LD 26;
      L     LD 22;
      A      [AR1,P#61.6];
      BLD   18;
      T     LD 22;
      TAK;
      T     LD 26;
      L     DIW [AR2,P#40.0];
      T     LW 30;
      OPN   DB [LW 30];
      L     DID [AR2,P#42.0];
      LAR1;
      L     LD 26;
      L     LD 22;
      =      [AR1,P#57.6];
      BLD   18;
      T     LD 22;
      TAK;
      T     LD 26;
      L     DIW [AR2,P#34.0];
      T     LW 30;
      OPN   DB [LW 30];
      L     DID [AR2,P#36.0];
      LAR1;
      L     LD 26;
      L     LD 22;
      L     D [AR1,P#28.0];
      L     1000;
      /D;
      BLD   18;
      T     LD 22;
      TAK;
      T     LD 26;
      L     DIW [AR2,P#40.0];
      T     LW 30;
      OPN   DB [LW 30];
      L     DID [AR2,P#42.0];
      LAR1;
      L     LD 26;
      L     LD 22;
      T     D [AR1,P#24.0];
      BLD   18;
      T     LD 22;
      TAK;
      T     LD 26;
      L     DIW [AR2,P#34.0];
      T     LW 30;
      OPN   DB [LW 30];
      L     DID [AR2,P#36.0];
      LAR1;
      L     LD 26;
      L     LD 22;
      L     D [AR1,P#32.0];
      L     1000;
      /D;
      BLD   18;
      T     LD 22;
      TAK;
      T     LD 26;
      L     DIW [AR2,P#40.0];
      T     LW 30;
      OPN   DB [LW 30];
      L     DID [AR2,P#42.0];
      LAR1;
      L     LD 26;
      L     LD 22;
      T     D [AR1,P#28.0];
      BLD   18;
      T     LD 22;
      TAK;
      T     LD 26;
      L     DIW [AR2,P#34.0];
      T     LW 30;
      OPN   DB [LW 30];
      L     DID [AR2,P#36.0];
      LAR1;
      L     LD 26;
      L     LD 22;
      A      [AR1,P#61.7];
      BLD   18;
      T     LD 22;
      TAK;
      T     LD 26;
      L     DIW [AR2,P#40.0];
      T     LW 30;
      OPN   DB [LW 30];
      L     DID [AR2,P#42.0];
      LAR1;
      L     LD 26;
      L     LD 22;
      =      [AR1,P#57.7];
      BLD   18;
      T     LD 22;
      TAK;
      T     LD 26;
      L     DIW [AR2,P#34.0];
      T     LW 30;
      OPN   DB [LW 30];
      L     DID [AR2,P#36.0];
      LAR1;
      L     LD 26;
      L     LD 22;
      L     D [AR1,P#44.0];
      BLD   18;
      T     LD 22;
      TAK;
      T     LD 26;
      L     DIW [AR2,P#40.0];
      T     LW 30;
      OPN   DB [LW 30];
      L     DID [AR2,P#42.0];
      LAR1;
      L     LD 26;
      L     LD 22;
      T     D [AR1,P#40.0];
      BLD   18;
      T     LD 22;
      TAK;
      T     LD 26;
      L     DIW [AR2,P#34.0];
      T     LW 30;
      OPN   DB [LW 30];
      L     DID [AR2,P#36.0];
      LAR1;
      L     LD 26;
      L     LD 22;
      L     D [AR1,P#48.0];
      BLD   18;
      T     LD 22;
      TAK;
      T     LD 26;
      L     DIW [AR2,P#40.0];
      T     LW 30;
      OPN   DB [LW 30];
      L     DID [AR2,P#42.0];
      LAR1;
      L     LD 26;
      L     LD 22;
      T     D [AR1,P#44.0];
      BLD   18;
      T     LD 22;
      TAK;
      T     LD 26;
      L     DIW [AR2,P#34.0];
      T     LW 30;
      OPN   DB [LW 30];
      L     DID [AR2,P#36.0];
      LAR1;
      L     LD 26;
      L     LD 22;
      L     D [AR1,P#36.0];
      BLD   18;
      T     LD 22;
      TAK;
      T     LD 26;
      L     DIW [AR2,P#40.0];
      T     LW 30;
      OPN   DB [LW 30];
      L     DID [AR2,P#42.0];
      LAR1;
      L     LD 26;
      L     LD 22;
      T     D [AR1,P#32.0];
      BLD   18;
      T     LD 22;
      TAK;
      T     LD 26;
      L     DIW [AR2,P#34.0];
      T     LW 30;
      OPN   DB [LW 30];
      L     DID [AR2,P#36.0];
      LAR1;
      L     LD 26;
      L     LD 22;
      A      [AR1,P#62.0];
      BLD   18;
      T     LD 22;
      TAK;
      T     LD 26;
      L     DIW [AR2,P#40.0];
      T     LW 30;
      OPN   DB [LW 30];
      L     DID [AR2,P#42.0];
      LAR1;
      L     LD 26;
      L     LD 22;
      =      [AR1,P#58.0];
      BLD   18;
      T     LD 22;
      TAK;
      T     LD 26;
      L     DIW [AR2,P#34.0];
      T     LW 30;
      OPN   DB [LW 30];
      L     DID [AR2,P#36.0];
      LAR1;
      L     LD 26;
      L     LD 22;
      L     D [AR1,P#40.0];
      BLD   18;
      T     LD 22;
      TAK;
      T     LD 26;
      L     DIW [AR2,P#40.0];
      T     LW 30;
      OPN   DB [LW 30];
      L     DID [AR2,P#42.0];
      LAR1;
      L     LD 26;
      L     LD 22;
      T     D [AR1,P#36.0];
      BLD   18;
      T     LD 22;
      TAK;
      T     LD 26;
      L     DIW [AR2,P#34.0];
      T     LW 30;
      OPN   DB [LW 30];
      L     DID [AR2,P#36.0];
      LAR1;
      L     LD 26;
      L     LD 22;
      A      [AR1,P#62.1];
      BLD   18;
      T     LD 22;
      TAK;
      T     LD 26;
      L     DIW [AR2,P#40.0];
      T     LW 30;
      OPN   DB [LW 30];
      L     DID [AR2,P#42.0];
      LAR1;
      L     LD 26;
      L     LD 22;
      =      [AR1,P#58.1];
      SET;
      BLD   18;
      T     LD 22;
      TAK;
      T     LD 26;
      L     DIW [AR2,P#40.0];
      T     LW 30;
      OPN   DB [LW 30];
      L     DID [AR2,P#42.0];
      LAR1;
      L     LD 26;
      L     LD 22;
      =      [AR1,P#62.0];
M011: BLD   18;
      T     LD 22;
      TAK;
      T     LD 26;
      L     DIW [AR2,P#34.0];
      T     LW 30;
      OPN   DB [LW 30];
      L     DID [AR2,P#36.0];
      LAR1;
      L     LD 26;
      L     LD 22;
      L     D [AR1,P#0.0];
      BLD   18;
      T     LD 22;
      TAK;
      T     LD 26;
      L     DIW [AR2,P#40.0];
      T     LW 30;
      OPN   DB [LW 30];
      L     DID [AR2,P#42.0];
      LAR1;
      L     LD 26;
      L     LD 22;
      T     D [AR1,P#0.0];
      BLD   18;
      T     LD 22;
      TAK;
      T     LD 26;
      L     DIW [AR2,P#34.0];
      T     LW 30;
      OPN   DB [LW 30];
      L     DID [AR2,P#36.0];
      LAR1;
      L     LD 26;
      L     LD 22;
      L     D [AR1,P#4.0];
      BLD   18;
      T     LD 22;
      TAK;
      T     LD 26;
      L     DIW [AR2,P#40.0];
      T     LW 30;
      OPN   DB [LW 30];
      L     DID [AR2,P#42.0];
      LAR1;
      L     LD 26;
      L     LD 22;
      T     D [AR1,P#4.0];
      BLD   18;
      T     LD 22;
      TAK;
      T     LD 26;
      L     DIW [AR2,P#40.0];
      T     LW 30;
      OPN   DB [LW 30];
      L     DID [AR2,P#42.0];
      LAR1;
      L     LD 26;
      L     LD 22;
      L     D [AR1,P#8.0];
      BLD   18;
      T     LD 22;
      TAK;
      T     LD 26;
      L     DIW [AR2,P#34.0];
      T     LW 30;
      OPN   DB [LW 30];
      L     DID [AR2,P#36.0];
      LAR1;
      L     LD 26;
      L     LD 22;
      T     D [AR1,P#8.0];
      BLD   18;
      T     LD 22;
      TAK;
      T     LD 26;
      L     DIW [AR2,P#34.0];
      T     LW 30;
      OPN   DB [LW 30];
      L     DID [AR2,P#36.0];
      LAR1;
      L     LD 26;
      L     LD 22;
      A      [AR1,P#61.0];
      BLD   18;
      T     LD 22;
      TAK;
      T     LD 26;
      L     DIW [AR2,P#34.0];
      T     LW 30;
      OPN   DB [LW 30];
      L     DID [AR2,P#36.0];
      LAR1;
      L     LD 26;
      L     LD 22;
      AN     [AR1,P#61.3];
      JC    M012;
      BLD   18;
      T     LD 22;
      TAK;
      T     LD 26;
      L     DIW [AR2,P#34.0];
      T     LW 30;
      OPN   DB [LW 30];
      L     DID [AR2,P#36.0];
      LAR1;
      L     LD 26;
      L     LD 22;
      L     D [AR1,P#16.0];
      BLD   18;
      T     LD 22;
      TAK;
      T     LD 26;
      L     DIW [AR2,P#40.0];
      T     LW 30;
      OPN   DB [LW 30];
      L     DID [AR2,P#42.0];
      LAR1;
      L     LD 26;
      L     LD 22;
      T     D [AR1,P#12.0];
      JU    M015;
M012: BLD   18;
      T     LD 22;
      TAK;
      T     LD 26;
      L     DIW [AR2,P#40.0];
      T     LW 30;
      OPN   DB [LW 30];
      L     DID [AR2,P#42.0];
      LAR1;
      L     LD 26;
      L     LD 22;
      L     D [AR1,P#12.0];
      BLD   18;
      T     LD 22;
      TAK;
      T     LD 26;
      L     DIW [AR2,P#34.0];
      T     LW 30;
      OPN   DB [LW 30];
      L     DID [AR2,P#36.0];
      LAR1;
      L     LD 26;
      L     LD 22;
      L     D [AR1,P#44.0];
      >R;
      JC    M013;
      BLD   18;
      T     LD 22;
      TAK;
      T     LD 26;
      L     DIW [AR2,P#40.0];
      T     LW 30;
      OPN   DB [LW 30];
      L     DID [AR2,P#42.0];
      LAR1;
      L     LD 26;
      L     LD 22;
      L     D [AR1,P#12.0];
      BLD   18;
      T     LD 22;
      TAK;
      T     LD 26;
      L     DIW [AR2,P#34.0];
      T     LW 30;
      OPN   DB [LW 30];
      L     DID [AR2,P#36.0];
      LAR1;
      L     LD 26;
      L     LD 22;
      L     D [AR1,P#48.0];
      <R;
      JC    M013;
      JU    M014;
M013: BLD   18;
      T     LD 22;
      TAK;
      T     LD 26;
      L     DIW [AR2,P#40.0];
      T     LW 30;
      OPN   DB [LW 30];
      L     DID [AR2,P#42.0];
      LAR1;
      L     LD 26;
      L     LD 22;
      T     D [AR1,P#12.0];
M014: BLD   18;
      T     LD 22;
      TAK;
      T     LD 26;
      L     DIW [AR2,P#40.0];
      T     LW 30;
      OPN   DB [LW 30];
      L     DID [AR2,P#42.0];
      LAR1;
      L     LD 26;
      L     LD 22;
      L     D [AR1,P#12.0];
      BLD   18;
      T     LD 22;
      TAK;
      T     LD 26;
      L     DIW [AR2,P#34.0];
      T     LW 30;
      OPN   DB [LW 30];
      L     DID [AR2,P#36.0];
      LAR1;
      L     LD 26;
      L     LD 22;
      T     D [AR1,P#16.0];
M015: NOP   0;
      A(;
      BLD   18;
      T     LD 22;
      TAK;
      T     LD 26;
      L     DIW [AR2,P#34.0];
      T     LW 30;
      OPN   DB [LW 30];
      L     DID [AR2,P#36.0];
      LAR1;
      L     LD 26;
      L     LD 22;
      A      [AR1,P#61.0];
      BLD   18;
      T     LD 22;
      TAK;
      T     LD 26;
      L     DIW [AR2,P#40.0];
      T     LW 30;
      OPN   DB [LW 30];
      L     DID [AR2,P#42.0];
      LAR1;
      L     LD 26;
      L     LD 22;
      AN     [AR1,P#57.0];
      O;
      BLD   18;
      T     LD 22;
      TAK;
      T     LD 26;
      L     DIW [AR2,P#34.0];
      T     LW 30;
      OPN   DB [LW 30];
      L     DID [AR2,P#36.0];
      LAR1;
      L     LD 26;
      L     LD 22;
      AN     [AR1,P#61.0];
      BLD   18;
      T     LD 22;
      TAK;
      T     LD 26;
      L     DIW [AR2,P#40.0];
      T     LW 30;
      OPN   DB [LW 30];
      L     DID [AR2,P#42.0];
      LAR1;
      L     LD 26;
      L     LD 22;
      A      [AR1,P#57.0];
      );
      =     L 0.0;
      BLD   16;
      =     L 28.0;
      L     DINO;
      T     LW 26;
      CDB;
      OPN   DI [LW 26];
      TAR2  LD 22;
      A     L 0.0;
      =     DIX [AR2,P#172.0];
      L     L#1000;
      T     DID [AR2,P#174.0];
      +AR2  P#172.0;
      UC    "TON";
      LAR2  LD 22;
      CDB;
      BLD   17;
      AN    DIX [AR2,P#178.0];
      JC    M016;
      BLD   18;
      T     LD 22;
      TAK;
      T     LD 26;
      L     DIW [AR2,P#34.0];
      T     LW 30;
      OPN   DB [LW 30];
      L     DID [AR2,P#36.0];
      LAR1;
      L     LD 26;
      L     LD 22;
      A      [AR1,P#61.0];
      BLD   18;
      T     LD 22;
      TAK;
      T     LD 26;
      L     DIW [AR2,P#40.0];
      T     LW 30;
      OPN   DB [LW 30];
      L     DID [AR2,P#42.0];
      LAR1;
      L     LD 26;
      L     LD 22;
      =      [AR1,P#57.0];
M016: BLD   18;
      T     LD 22;
      TAK;
      T     LD 26;
      L     DIW [AR2,P#40.0];
      T     LW 30;
      OPN   DB [LW 30];
      L     DID [AR2,P#42.0];
      LAR1;
      L     LD 26;
      L     LD 22;
      A      [AR1,P#57.0];
      =     DIX [AR2,P#32.1];
      A(;
      BLD   18;
      T     LD 22;
      TAK;
      T     LD 26;
      L     DIW [AR2,P#34.0];
      T     LW 30;
      OPN   DB [LW 30];
      L     DID [AR2,P#36.0];
      LAR1;
      L     LD 26;
      L     LD 22;
      A      [AR1,P#61.1];
      BLD   18;
      T     LD 22;
      TAK;
      T     LD 26;
      L     DIW [AR2,P#40.0];
      T     LW 30;
      OPN   DB [LW 30];
      L     DID [AR2,P#42.0];
      LAR1;
      L     LD 26;
      L     LD 22;
      AN     [AR1,P#57.1];
      O;
      BLD   18;
      T     LD 22;
      TAK;
      T     LD 26;
      L     DIW [AR2,P#34.0];
      T     LW 30;
      OPN   DB [LW 30];
      L     DID [AR2,P#36.0];
      LAR1;
      L     LD 26;
      L     LD 22;
      AN     [AR1,P#61.1];
      BLD   18;
      T     LD 22;
      TAK;
      T     LD 26;
      L     DIW [AR2,P#40.0];
      T     LW 30;
      OPN   DB [LW 30];
      L     DID [AR2,P#42.0];
      LAR1;
      L     LD 26;
      L     LD 22;
      A      [AR1,P#57.1];
      );
      =     L 0.1;
      BLD   16;
      =     L 28.0;
      L     DINO;
      T     LW 26;
      CDB;
      OPN   DI [LW 26];
      TAR2  LD 22;
      A     L 0.1;
      =     DIX [AR2,P#194.0];
      L     L#1000;
      T     DID [AR2,P#196.0];
      +AR2  P#194.0;
      UC    "TON";
      LAR2  LD 22;
      CDB;
      BLD   17;
      AN    DIX [AR2,P#200.0];
      JC    M017;
      BLD   18;
      T     LD 22;
      TAK;
      T     LD 26;
      L     DIW [AR2,P#34.0];
      T     LW 30;
      OPN   DB [LW 30];
      L     DID [AR2,P#36.0];
      LAR1;
      L     LD 26;
      L     LD 22;
      A      [AR1,P#61.1];
      BLD   18;
      T     LD 22;
      TAK;
      T     LD 26;
      L     DIW [AR2,P#40.0];
      T     LW 30;
      OPN   DB [LW 30];
      L     DID [AR2,P#42.0];
      LAR1;
      L     LD 26;
      L     LD 22;
      =      [AR1,P#57.1];
M017: BLD   18;
      T     LD 22;
      TAK;
      T     LD 26;
      L     DIW [AR2,P#40.0];
      T     LW 30;
      OPN   DB [LW 30];
      L     DID [AR2,P#42.0];
      LAR1;
      L     LD 26;
      L     LD 22;
      A      [AR1,P#57.1];
      =     DIX [AR2,P#32.0];
      BLD   18;
      T     LD 22;
      TAK;
      T     LD 26;
      L     DIW [AR2,P#40.0];
      T     LW 30;
      OPN   DB [LW 30];
      L     DID [AR2,P#42.0];
      LAR1;
      L     LD 26;
      L     LD 22;
      L     D [AR1,P#16.0];
      L     1.000000e-05;
      <R;
      JC    M018;
      BLD   18;
      T     LD 22;
      TAK;
      T     LD 26;
      L     DIW [AR2,P#40.0];
      T     LW 30;
      OPN   DB [LW 30];
      L     DID [AR2,P#42.0];
      LAR1;
      L     LD 26;
      L     LD 22;
      L     D [AR1,P#16.0];
      L     2.000000e+01;
      >R;
      JC    M018;
      JU    M019;
M018: BLD   18;
      T     LD 22;
      TAK;
      T     LD 26;
      L     DIW [AR2,P#40.0];
      T     LW 30;
      OPN   DB [LW 30];
      L     DID [AR2,P#42.0];
      LAR1;
      L     LD 26;
      L     LD 22;
      T     D [AR1,P#16.0];
M019: BLD   18;
      T     LD 22;
      TAK;
      T     LD 26;
      L     DIW [AR2,P#40.0];
      T     LW 30;
      OPN   DB [LW 30];
      L     DID [AR2,P#42.0];
      LAR1;
      L     LD 26;
      L     LD 22;
      L     D [AR1,P#16.0];
      BLD   18;
      T     LD 22;
      TAK;
      T     LD 26;
      L     DIW [AR2,P#34.0];
      T     LW 30;
      OPN   DB [LW 30];
      L     DID [AR2,P#36.0];
      LAR1;
      L     LD 26;
      L     LD 22;
      T     D [AR1,P#20.0];
      BLD   18;
      T     LD 22;
      TAK;
      T     LD 26;
      L     DIW [AR2,P#40.0];
      T     LW 30;
      OPN   DB [LW 30];
      L     DID [AR2,P#42.0];
      LAR1;
      L     LD 26;
      L     LD 22;
      A      [AR1,P#57.4];
      BLD   18;
      T     LD 22;
      TAK;
      T     LD 26;
      L     DIW [AR2,P#34.0];
      T     LW 30;
      OPN   DB [LW 30];
      L     DID [AR2,P#36.0];
      LAR1;
      L     LD 26;
      L     LD 22;
      =      [AR1,P#61.4];
      BLD   18;
      T     LD 22;
      TAK;
      T     LD 26;
      L     DIW [AR2,P#40.0];
      T     LW 30;
      OPN   DB [LW 30];
      L     DID [AR2,P#42.0];
      LAR1;
      L     LD 26;
      L     LD 22;
      A      [AR1,P#57.5];
      BLD   18;
      T     LD 22;
      TAK;
      T     LD 26;
      L     DIW [AR2,P#34.0];
      T     LW 30;
      OPN   DB [LW 30];
      L     DID [AR2,P#36.0];
      LAR1;
      L     LD 26;
      L     LD 22;
      =      [AR1,P#61.5];
      BLD   18;
      T     LD 22;
      TAK;
      T     LD 26;
      L     DIW [AR2,P#40.0];
      T     LW 30;
      OPN   DB [LW 30];
      L     DID [AR2,P#42.0];
      LAR1;
      L     LD 26;
      L     LD 22;
      L     D [AR1,P#20.0];
      L     1000;
      *D;
      L     T#0MS;
      <D;
      JC    M020;
      BLD   18;
      T     LD 22;
      TAK;
      T     LD 26;
      L     DIW [AR2,P#40.0];
      T     LW 30;
      OPN   DB [LW 30];
      L     DID [AR2,P#42.0];
      LAR1;
      L     LD 26;
      L     LD 22;
      L     D [AR1,P#20.0];
      L     1000;
      *D;
      L     T#1H;
      >D;
      JC    M020;
      JU    M021;
M020: L     1000;
      /D;
      BLD   18;
      T     LD 22;
      TAK;
      T     LD 26;
      L     DIW [AR2,P#40.0];
      T     LW 30;
      OPN   DB [LW 30];
      L     DID [AR2,P#42.0];
      LAR1;
      L     LD 26;
      L     LD 22;
      T     D [AR1,P#20.0];
M021: BLD   18;
      T     LD 22;
      TAK;
      T     LD 26;
      L     DIW [AR2,P#40.0];
      T     LW 30;
      OPN   DB [LW 30];
      L     DID [AR2,P#42.0];
      LAR1;
      L     LD 26;
      L     LD 22;
      L     D [AR1,P#20.0];
      L     1000;
      *D;
      BLD   18;
      T     LD 22;
      TAK;
      T     LD 26;
      L     DIW [AR2,P#34.0];
      T     LW 30;
      OPN   DB [LW 30];
      L     DID [AR2,P#36.0];
      LAR1;
      L     LD 26;
      L     LD 22;
      T     D [AR1,P#24.0];
      BLD   18;
      T     LD 22;
      TAK;
      T     LD 26;
      L     DIW [AR2,P#40.0];
      T     LW 30;
      OPN   DB [LW 30];
      L     DID [AR2,P#42.0];
      LAR1;
      L     LD 26;
      L     LD 22;
      A      [AR1,P#57.6];
      BLD   18;
      T     LD 22;
      TAK;
      T     LD 26;
      L     DIW [AR2,P#34.0];
      T     LW 30;
      OPN   DB [LW 30];
      L     DID [AR2,P#36.0];
      LAR1;
      L     LD 26;
      L     LD 22;
      =      [AR1,P#61.6];
      BLD   18;
      T     LD 22;
      TAK;
      T     LD 26;
      L     DIW [AR2,P#40.0];
      T     LW 30;
      OPN   DB [LW 30];
      L     DID [AR2,P#42.0];
      LAR1;
      L     LD 26;
      L     LD 22;
      L     D [AR1,P#24.0];
      L     1000;
      *D;
      L     T#0MS;
      <D;
      JC    M022;
      BLD   18;
      T     LD 22;
      TAK;
      T     LD 26;
      L     DIW [AR2,P#40.0];
      T     LW 30;
      OPN   DB [LW 30];
      L     DID [AR2,P#42.0];
      LAR1;
      L     LD 26;
      L     LD 22;
      L     D [AR1,P#24.0];
      L     1000;
      *D;
      L     T#10M;
      >D;
      JC    M022;
      JU    M023;
M022: L     1000;
      /D;
      BLD   18;
      T     LD 22;
      TAK;
      T     LD 26;
      L     DIW [AR2,P#40.0];
      T     LW 30;
      OPN   DB [LW 30];
      L     DID [AR2,P#42.0];
      LAR1;
      L     LD 26;
      L     LD 22;
      T     D [AR1,P#24.0];
M023: BLD   18;
      T     LD 22;
      TAK;
      T     LD 26;
      L     DIW [AR2,P#40.0];
      T     LW 30;
      OPN   DB [LW 30];
      L     DID [AR2,P#42.0];
      LAR1;
      L     LD 26;
      L     LD 22;
      L     D [AR1,P#24.0];
      L     1000;
      *D;
      BLD   18;
      T     LD 22;
      TAK;
      T     LD 26;
      L     DIW [AR2,P#34.0];
      T     LW 30;
      OPN   DB [LW 30];
      L     DID [AR2,P#36.0];
      LAR1;
      L     LD 26;
      L     LD 22;
      T     D [AR1,P#28.0];
      BLD   18;
      T     LD 22;
      TAK;
      T     LD 26;
      L     DIW [AR2,P#40.0];
      T     LW 30;
      OPN   DB [LW 30];
      L     DID [AR2,P#42.0];
      LAR1;
      L     LD 26;
      L     LD 22;
      L     D [AR1,P#28.0];
      L     1000;
      *D;
      L     T#0MS;
      <D;
      JC    M024;
      BLD   18;
      T     LD 22;
      TAK;
      T     LD 26;
      L     DIW [AR2,P#40.0];
      T     LW 30;
      OPN   DB [LW 30];
      L     DID [AR2,P#42.0];
      LAR1;
      L     LD 26;
      L     LD 22;
      L     D [AR1,P#28.0];
      L     1000;
      *D;
      L     T#5M;
      >D;
      JC    M024;
      JU    M025;
M024: L     1000;
      /D;
      BLD   18;
      T     LD 22;
      TAK;
      T     LD 26;
      L     DIW [AR2,P#40.0];
      T     LW 30;
      OPN   DB [LW 30];
      L     DID [AR2,P#42.0];
      LAR1;
      L     LD 26;
      L     LD 22;
      T     D [AR1,P#28.0];
M025: BLD   18;
      T     LD 22;
      TAK;
      T     LD 26;
      L     DIW [AR2,P#40.0];
      T     LW 30;
      OPN   DB [LW 30];
      L     DID [AR2,P#42.0];
      LAR1;
      L     LD 26;
      L     LD 22;
      L     D [AR1,P#28.0];
      L     1000;
      *D;
      BLD   18;
      T     LD 22;
      TAK;
      T     LD 26;
      L     DIW [AR2,P#34.0];
      T     LW 30;
      OPN   DB [LW 30];
      L     DID [AR2,P#36.0];
      LAR1;
      L     LD 26;
      L     LD 22;
      T     D [AR1,P#32.0];
      BLD   18;
      T     LD 22;
      TAK;
      T     LD 26;
      L     DIW [AR2,P#40.0];
      T     LW 30;
      OPN   DB [LW 30];
      L     DID [AR2,P#42.0];
      LAR1;
      L     LD 26;
      L     LD 22;
      A      [AR1,P#57.7];
      BLD   18;
      T     LD 22;
      TAK;
      T     LD 26;
      L     DIW [AR2,P#34.0];
      T     LW 30;
      OPN   DB [LW 30];
      L     DID [AR2,P#36.0];
      LAR1;
      L     LD 26;
      L     LD 22;
      =      [AR1,P#61.7];
      BLD   18;
      T     LD 22;
      TAK;
      T     LD 26;
      L     DIW [AR2,P#40.0];
      T     LW 30;
      OPN   DB [LW 30];
      L     DID [AR2,P#42.0];
      LAR1;
      L     LD 26;
      L     LD 22;
      L     D [AR1,P#40.0];
      BLD   18;
      T     LD 22;
      TAK;
      T     LD 26;
      L     DIW [AR2,P#40.0];
      T     LW 30;
      OPN   DB [LW 30];
      L     DID [AR2,P#42.0];
      LAR1;
      L     LD 26;
      L     LD 22;
      L     D [AR1,P#44.0];
      <R;
      JC    M026;
      BLD   18;
      T     LD 22;
      TAK;
      T     LD 26;
      L     DIW [AR2,P#40.0];
      T     LW 30;
      OPN   DB [LW 30];
      L     DID [AR2,P#42.0];
      LAR1;
      L     LD 26;
      L     LD 22;
      L     D [AR1,P#40.0];
      L     1.000000e+02;
      >R;
      JC    M026;
      JU    M027;
M026: BLD   18;
      T     LD 22;
      TAK;
      T     LD 26;
      L     DIW [AR2,P#40.0];
      T     LW 30;
      OPN   DB [LW 30];
      L     DID [AR2,P#42.0];
      LAR1;
      L     LD 26;
      L     LD 22;
      T     D [AR1,P#40.0];
M027: BLD   18;
      T     LD 22;
      TAK;
      T     LD 26;
      L     DIW [AR2,P#40.0];
      T     LW 30;
      OPN   DB [LW 30];
      L     DID [AR2,P#42.0];
      LAR1;
      L     LD 26;
      L     LD 22;
      L     D [AR1,P#40.0];
      BLD   18;
      T     LD 22;
      TAK;
      T     LD 26;
      L     DIW [AR2,P#34.0];
      T     LW 30;
      OPN   DB [LW 30];
      L     DID [AR2,P#36.0];
      LAR1;
      L     LD 26;
      L     LD 22;
      T     D [AR1,P#44.0];
      BLD   18;
      T     LD 22;
      TAK;
      T     LD 26;
      L     DIW [AR2,P#40.0];
      T     LW 30;
      OPN   DB [LW 30];
      L     DID [AR2,P#42.0];
      LAR1;
      L     LD 26;
      L     LD 22;
      L     D [AR1,P#44.0];
      L     0.000000e+00;
      <R;
      JC    M028;
      BLD   18;
      T     LD 22;
      TAK;
      T     LD 26;
      L     DIW [AR2,P#40.0];
      T     LW 30;
      OPN   DB [LW 30];
      L     DID [AR2,P#42.0];
      LAR1;
      L     LD 26;
      L     LD 22;
      L     D [AR1,P#44.0];
      BLD   18;
      T     LD 22;
      TAK;
      T     LD 26;
      L     DIW [AR2,P#40.0];
      T     LW 30;
      OPN   DB [LW 30];
      L     DID [AR2,P#42.0];
      LAR1;
      L     LD 26;
      L     LD 22;
      L     D [AR1,P#40.0];
      >R;
      JC    M028;
      JU    M029;
M028: BLD   18;
      T     LD 22;
      TAK;
      T     LD 26;
      L     DIW [AR2,P#40.0];
      T     LW 30;
      OPN   DB [LW 30];
      L     DID [AR2,P#42.0];
      LAR1;
      L     LD 26;
      L     LD 22;
      T     D [AR1,P#44.0];
M029: BLD   18;
      T     LD 22;
      TAK;
      T     LD 26;
      L     DIW [AR2,P#40.0];
      T     LW 30;
      OPN   DB [LW 30];
      L     DID [AR2,P#42.0];
      LAR1;
      L     LD 26;
      L     LD 22;
      L     D [AR1,P#44.0];
      BLD   18;
      T     LD 22;
      TAK;
      T     LD 26;
      L     DIW [AR2,P#34.0];
      T     LW 30;
      OPN   DB [LW 30];
      L     DID [AR2,P#36.0];
      LAR1;
      L     LD 26;
      L     LD 22;
      T     D [AR1,P#48.0];
      L     DID [AR2,P#24.0];
      BLD   18;
      T     LD 22;
      TAK;
      T     LD 26;
      L     DIW [AR2,P#34.0];
      T     LW 30;
      OPN   DB [LW 30];
      L     DID [AR2,P#36.0];
      LAR1;
      L     LD 26;
      L     LD 22;
      AN     [AR1,P#62.0];
      JC    M030;
      BLD   18;
      T     LD 22;
      TAK;
      T     LD 26;
      L     DIW [AR2,P#40.0];
      T     LW 30;
      OPN   DB [LW 30];
      L     DID [AR2,P#42.0];
      LAR1;
      L     LD 26;
      L     LD 22;
      L     D [AR1,P#32.0];
      L     T#10MS;
      <D;
      JC    M030;
      BLD   18;
      T     LD 22;
      TAK;
      T     LD 26;
      L     DIW [AR2,P#40.0];
      T     LW 30;
      OPN   DB [LW 30];
      L     DID [AR2,P#42.0];
      LAR1;
      L     LD 26;
      L     LD 22;
      L     D [AR1,P#32.0];
      L     T#1M;
      >D;
      JC    M030;
      JU    M031;
M030: BLD   18;
      T     LD 22;
      TAK;
      T     LD 26;
      L     DIW [AR2,P#40.0];
      T     LW 30;
      OPN   DB [LW 30];
      L     DID [AR2,P#42.0];
      LAR1;
      L     LD 26;
      L     LD 22;
      T     D [AR1,P#32.0];
M031: BLD   18;
      T     LD 22;
      TAK;
      T     LD 26;
      L     DIW [AR2,P#40.0];
      T     LW 30;
      OPN   DB [LW 30];
      L     DID [AR2,P#42.0];
      LAR1;
      L     LD 26;
      L     LD 22;
      L     D [AR1,P#32.0];
      BLD   18;
      T     LD 22;
      TAK;
      T     LD 26;
      L     DIW [AR2,P#34.0];
      T     LW 30;
      OPN   DB [LW 30];
      L     DID [AR2,P#36.0];
      LAR1;
      L     LD 26;
      L     LD 22;
      T     D [AR1,P#36.0];
      BLD   18;
      T     LD 22;
      TAK;
      T     LD 26;
      L     DIW [AR2,P#40.0];
      T     LW 30;
      OPN   DB [LW 30];
      L     DID [AR2,P#42.0];
      LAR1;
      L     LD 26;
      L     LD 22;
      A      [AR1,P#58.0];
      BLD   18;
      T     LD 22;
      TAK;
      T     LD 26;
      L     DIW [AR2,P#34.0];
      T     LW 30;
      OPN   DB [LW 30];
      L     DID [AR2,P#36.0];
      LAR1;
      L     LD 26;
      L     LD 22;
      =      [AR1,P#62.0];
      L     DID [AR2,P#24.0];
      BLD   18;
      T     LD 22;
      TAK;
      T     LD 26;
      L     DIW [AR2,P#34.0];
      T     LW 30;
      OPN   DB [LW 30];
      L     DID [AR2,P#36.0];
      LAR1;
      L     LD 26;
      L     LD 22;
      AN     [AR1,P#62.1];
      JC    M032;
      BLD   18;
      T     LD 22;
      TAK;
      T     LD 26;
      L     DIW [AR2,P#40.0];
      T     LW 30;
      OPN   DB [LW 30];
      L     DID [AR2,P#42.0];
      LAR1;
      L     LD 26;
      L     LD 22;
      L     D [AR1,P#36.0];
      L     T#10MS;
      <D;
      JC    M032;
      BLD   18;
      T     LD 22;
      TAK;
      T     LD 26;
      L     DIW [AR2,P#40.0];
      T     LW 30;
      OPN   DB [LW 30];
      L     DID [AR2,P#42.0];
      LAR1;
      L     LD 26;
      L     LD 22;
      L     D [AR1,P#36.0];
      L     T#1M;
      >D;
      JC    M032;
      JU    M033;
M032: BLD   18;
      T     LD 22;
      TAK;
      T     LD 26;
      L     DIW [AR2,P#40.0];
      T     LW 30;
      OPN   DB [LW 30];
      L     DID [AR2,P#42.0];
      LAR1;
      L     LD 26;
      L     LD 22;
      T     D [AR1,P#36.0];
M033: BLD   18;
      T     LD 22;
      TAK;
      T     LD 26;
      L     DIW [AR2,P#40.0];
      T     LW 30;
      OPN   DB [LW 30];
      L     DID [AR2,P#42.0];
      LAR1;
      L     LD 26;
      L     LD 22;
      L     D [AR1,P#36.0];
      BLD   18;
      T     LD 22;
      TAK;
      T     LD 26;
      L     DIW [AR2,P#34.0];
      T     LW 30;
      OPN   DB [LW 30];
      L     DID [AR2,P#36.0];
      LAR1;
      L     LD 26;
      L     LD 22;
      T     D [AR1,P#40.0];
      BLD   18;
      T     LD 22;
      TAK;
      T     LD 26;
      L     DIW [AR2,P#40.0];
      T     LW 30;
      OPN   DB [LW 30];
      L     DID [AR2,P#42.0];
      LAR1;
      L     LD 26;
      L     LD 22;
      A      [AR1,P#58.1];
      BLD   18;
      T     LD 22;
      TAK;
      T     LD 26;
      L     DIW [AR2,P#34.0];
      T     LW 30;
      OPN   DB [LW 30];
      L     DID [AR2,P#36.0];
      LAR1;
      L     LD 26;
      L     LD 22;
      =      [AR1,P#62.1];
      BLD   18;
      T     LD 22;
      TAK;
      T     LD 26;
      L     DIW [AR2,P#34.0];
      T     LW 30;
      OPN   DB [LW 30];
      L     DID [AR2,P#36.0];
      LAR1;
      L     LD 26;
      L     LD 22;
      A      [AR1,P#61.2];
      BLD   18;
      T     LD 22;
      TAK;
      T     LD 26;
      L     DIW [AR2,P#40.0];
      T     LW 30;
      OPN   DB [LW 30];
      L     DID [AR2,P#42.0];
      LAR1;
      L     LD 26;
      L     LD 22;
      =      [AR1,P#57.2];
      BLD   18;
      T     LD 22;
      TAK;
      T     LD 26;
      L     DIW [AR2,P#34.0];
      T     LW 30;
      OPN   DB [LW 30];
      L     DID [AR2,P#36.0];
      LAR1;
      L     LD 26;
      L     LD 22;
      A      [AR1,P#61.3];
      BLD   18;
      T     LD 22;
      TAK;
      T     LD 26;
      L     DIW [AR2,P#40.0];
      T     LW 30;
      OPN   DB [LW 30];
      L     DID [AR2,P#42.0];
      LAR1;
      L     LD 26;
      L     LD 22;
      =      [AR1,P#57.3];
      BLD   18;
      T     LD 22;
      TAK;
      T     LD 26;
      L     DIW [AR2,P#34.0];
      T     LW 30;
      OPN   DB [LW 30];
      L     DID [AR2,P#36.0];
      LAR1;
      L     LD 26;
      L     LD 22;
      L     B [AR1,P#60.0];
      BLD   18;
      T     LD 22;
      TAK;
      T     LD 26;
      L     DIW [AR2,P#40.0];
      T     LW 30;
      OPN   DB [LW 30];
      L     DID [AR2,P#42.0];
      LAR1;
      L     LD 26;
      L     LD 22;
      T     B [AR1,P#56.0];
M034: NOP   0;
      BLD   18;
      T     LD 22;
      TAK;
      T     LD 26;
      L     DIW [AR2,P#34.0];
      T     LW 30;
      OPN   DB [LW 30];
      L     DID [AR2,P#36.0];
      LAR1;
      L     LD 26;
      L     LD 22;
      L     D [AR1,P#52.0];
      BLD   18;
      T     LD 22;
      TAK;
      T     LD 26;
      L     DIW [AR2,P#34.0];
      T     LW 30;
      OPN   DB [LW 30];
      L     DID [AR2,P#36.0];
      LAR1;
      L     LD 26;
      L     LD 22;
      L     D [AR1,P#48.0];
      <R;
      JC    M035;
      BLD   18;
      T     LD 22;
      TAK;
      T     LD 26;
      L     DIW [AR2,P#34.0];
      T     LW 30;
      OPN   DB [LW 30];
      L     DID [AR2,P#36.0];
      LAR1;
      L     LD 26;
      L     LD 22;
      L     D [AR1,P#52.0];
      BLD   18;
      T     LD 22;
      TAK;
      T     LD 26;
      L     DIW [AR2,P#34.0];
      T     LW 30;
      OPN   DB [LW 30];
      L     DID [AR2,P#36.0];
      LAR1;
      L     LD 26;
      L     LD 22;
      L     D [AR1,P#44.0];
      >R;
      JC    M035;
      JU    M036;
M035: BLD   18;
      T     LD 22;
      TAK;
      T     LD 26;
      L     DIW [AR2,P#34.0];
      T     LW 30;
      OPN   DB [LW 30];
      L     DID [AR2,P#36.0];
      LAR1;
      L     LD 26;
      L     LD 22;
      T     D [AR1,P#52.0];
M036: NOP   0;
      BLD   18;
      T     LD 22;
      TAK;
      T     LD 26;
      L     DIW [AR2,P#34.0];
      T     LW 30;
      OPN   DB [LW 30];
      L     DID [AR2,P#36.0];
      LAR1;
      L     LD 26;
      L     LD 22;
      L     D [AR1,P#56.0];
      L     0.000000e+00;
      <R;
      JC    M037;
      BLD   18;
      T     LD 22;
      TAK;
      T     LD 26;
      L     DIW [AR2,P#34.0];
      T     LW 30;
      OPN   DB [LW 30];
      L     DID [AR2,P#36.0];
      LAR1;
      L     LD 26;
      L     LD 22;
      L     D [AR1,P#56.0];
      L     1.000000e+02;
      >R;
      JC    M037;
      JU    M038;
M037: BLD   18;
      T     LD 22;
      TAK;
      T     LD 26;
      L     DIW [AR2,P#34.0];
      T     LW 30;
      OPN   DB [LW 30];
      L     DID [AR2,P#36.0];
      LAR1;
      L     LD 26;
      L     LD 22;
      T     D [AR1,P#56.0];
M038: NOP   0;
NETWORK
TITLE =
      BLD   18;
      T     LD 22;
      TAK;
      T     LD 26;
      L     DIW [AR2,P#34.0];
      T     LW 30;
      OPN   DB [LW 30];
      L     DID [AR2,P#36.0];
      LAR1;
      L     LD 26;
      L     LD 22;
      AN     [AR1,P#61.5];
      JC    M039;
      BLD   18;
      T     LD 22;
      TAK;
      T     LD 26;
      L     DIW [AR2,P#34.0];
      T     LW 30;
      OPN   DB [LW 30];
      L     DID [AR2,P#36.0];
      LAR1;
      L     LD 26;
      L     LD 22;
      L     D [AR1,P#20.0];
      L     -1.000000e+00;
      *R;
      JU    M040;
M039: BLD   18;
      T     LD 22;
      TAK;
      T     LD 26;
      L     DIW [AR2,P#34.0];
      T     LW 30;
      OPN   DB [LW 30];
      L     DID [AR2,P#36.0];
      LAR1;
      L     LD 26;
      L     LD 22;
      L     D [AR1,P#20.0];
M040: T     LD 2;
      BLD   18;
      T     LD 22;
      TAK;
      T     LD 26;
      L     DIW [AR2,P#34.0];
      T     LW 30;
      OPN   DB [LW 30];
      L     DID [AR2,P#36.0];
      LAR1;
      L     LD 26;
      L     LD 22;
      AN     [AR1,P#61.1];
      JC    M041;
      BLD   18;
      T     LD 22;
      TAK;
      T     LD 26;
      L     DIW [AR2,P#34.0];
      T     LW 30;
      OPN   DB [LW 30];
      L     DID [AR2,P#36.0];
      LAR1;
      L     LD 26;
      L     LD 22;
      L     D [AR1,P#4.0];
      JU    M042;
M041: BLD   18;
      T     LD 22;
      TAK;
      T     LD 26;
      L     DIW [AR2,P#34.0];
      T     LW 30;
      OPN   DB [LW 30];
      L     DID [AR2,P#36.0];
      LAR1;
      L     LD 26;
      L     LD 22;
      L     D [AR1,P#8.0];
M042: BLD   18;
      T     LD 22;
      TAK;
      T     LD 26;
      L     DIW [AR2,P#34.0];
      T     LW 30;
      OPN   DB [LW 30];
      L     DID [AR2,P#36.0];
      LAR1;
      L     LD 26;
      L     LD 22;
      T     D [AR1,P#12.0];
NETWORK
TITLE =
      L     DID [AR2,P#118.0];
      L     DW#16#FFFFFFFF;
      ==D;
      =     L 16.0;
NETWORK
TITLE =
      BLD   18;
      T     LD 22;
      TAK;
      T     LD 26;
      L     DIW [AR2,P#34.0];
      T     LW 30;
      OPN   DB [LW 30];
      L     DID [AR2,P#36.0];
      LAR1;
      L     LD 26;
      L     LD 22;
      O      [AR1,P#61.2];
      BLD   18;
      T     LD 22;
      TAK;
      T     LD 26;
      L     DIW [AR2,P#34.0];
      T     LW 30;
      OPN   DB [LW 30];
      L     DID [AR2,P#36.0];
      LAR1;
      L     LD 26;
      L     LD 22;
      O      [AR1,P#61.3];
      BLD   18;
      T     LD 22;
      TAK;
      T     LD 26;
      L     DIW [AR2,P#34.0];
      T     LW 30;
      OPN   DB [LW 30];
      L     DID [AR2,P#36.0];
      LAR1;
      L     LD 26;
      L     LD 22;
      O      [AR1,P#61.0];
      =     L 16.1;
      BLD   18;
      T     LD 22;
      TAK;
      T     LD 26;
      L     DIW [AR2,P#34.0];
      T     LW 30;
      OPN   DB [LW 30];
      L     DID [AR2,P#36.0];
      LAR1;
      L     LD 26;
      L     LD 22;
      A      [AR1,P#61.3];
      BLD   18;
      T     LD 22;
      TAK;
      T     LD 26;
      L     DIW [AR2,P#34.0];
      T     LW 30;
      OPN   DB [LW 30];
      L     DID [AR2,P#36.0];
      LAR1;
      L     LD 26;
      L     LD 22;
      L     D [AR1,P#56.0];
      JC    M043;
      BLD   18;
      T     LD 22;
      TAK;
      T     LD 26;
      L     DIW [AR2,P#34.0];
      T     LW 30;
      OPN   DB [LW 30];
      L     DID [AR2,P#36.0];
      LAR1;
      L     LD 26;
      L     LD 22;
      A      [AR1,P#61.0];
      BLD   18;
      T     LD 22;
      TAK;
      T     LD 26;
      L     DIW [AR2,P#34.0];
      T     LW 30;
      OPN   DB [LW 30];
      L     DID [AR2,P#36.0];
      LAR1;
      L     LD 26;
      L     LD 22;
      L     D [AR1,P#16.0];
      JC    M043;
      BLD   18;
      T     LD 22;
      TAK;
      T     LD 26;
      L     DIW [AR2,P#34.0];
      T     LW 30;
      OPN   DB [LW 30];
      L     DID [AR2,P#36.0];
      LAR1;
      L     LD 26;
      L     LD 22;
      A      [AR1,P#61.2];
      BLD   18;
      T     LD 22;
      TAK;
      T     LD 26;
      L     DIW [AR2,P#34.0];
      T     LW 30;
      OPN   DB [LW 30];
      L     DID [AR2,P#36.0];
      LAR1;
      L     LD 26;
      L     LD 22;
      L     D [AR1,P#52.0];
      JC    M043;
      L     0.000000e+00;
M043: T     LD 18;
NETWORK
TITLE =
      BLD   14;
      =     L 28.0;
      L     DINO;
      T     LW 26;
      CDB;
      OPN   DI [LW 26];
      TAR2  LD 22;
      A     L 16.0;
      =     DIX [AR2,P#46.0];
      A     L 16.1;
      =     DIX [AR2,P#46.1];
      A     L 6.0;
      =     DIX [AR2,P#46.2];
      L     DBW [AR2,P#34.0];
      T     LW 29;
      OPN   DI [LW 29];
      L     DBD [AR2,P#36.0];
      LAR1;
      CDB;
      A      [AR1,P#61.4];
      CDB;
      OPN   DI [LW 26];
      =     DIX [AR2,P#46.3];
      L     DBW [AR2,P#34.0];
      T     LW 31;
      OPN   DI [LW 31];
      L     DBD [AR2,P#36.0];
      LAR1;
      CDB;
      A      [AR1,P#61.6];
      CDB;
      OPN   DI [LW 26];
      =     DIX [AR2,P#46.4];
      A     L 6.0;
      =     DIX [AR2,P#46.5];
      A     L 6.0;
      =     DIX [AR2,P#46.6];
      L     DBW [AR2,P#34.0];
      T     LW 33;
      OPN   DI [LW 33];
      L     DBD [AR2,P#36.0];
      LAR1;
      CDB;
      A      [AR1,P#61.7];
      CDB;
      OPN   DI [LW 26];
      =     DIX [AR2,P#46.7];
      L     L#1000;
      T     DID [AR2,P#48.0];
      L     DBW [AR2,P#34.0];
      T     LW 35;
      OPN   DI [LW 35];
      L     DBD [AR2,P#36.0];
      LAR1;
      CDB;
      L     D [AR1,P#12.0];
      CDB;
      OPN   DI [LW 26];
      T     DID [AR2,P#52.0];
      L     DBW [AR2,P#34.0];
      T     LW 37;
      OPN   DI [LW 37];
      L     DBD [AR2,P#36.0];
      LAR1;
      CDB;
      L     D [AR1,P#0.0];
      CDB;
      OPN   DI [LW 26];
      T     DID [AR2,P#56.0];
      L     0;
      T     DIW [AR2,P#60.0];
      L     LD 18;
      T     DID [AR2,P#62.0];
      L     LD 2;
      T     DID [AR2,P#66.0];
      L     DBW [AR2,P#34.0];
      T     LW 39;
      OPN   DI [LW 39];
      L     DBD [AR2,P#36.0];
      LAR1;
      CDB;
      L     D [AR1,P#24.0];
      CDB;
      OPN   DI [LW 26];
      T     DID [AR2,P#70.0];
      L     DBW [AR2,P#34.0];
      T     LW 41;
      OPN   DI [LW 41];
      L     DBD [AR2,P#36.0];
      LAR1;
      CDB;
      L     D [AR1,P#28.0];
      CDB;
      OPN   DI [LW 26];
      T     DID [AR2,P#74.0];
      L     DBW [AR2,P#34.0];
      T     LW 43;
      OPN   DI [LW 43];
      L     DBD [AR2,P#36.0];
      LAR1;
      CDB;
      L     D [AR1,P#32.0];
      CDB;
      OPN   DI [LW 26];
      T     DID [AR2,P#78.0];
      L     L#0;
      T     DID [AR2,P#82.0];
      L     DBW [AR2,P#34.0];
      T     LW 45;
      OPN   DI [LW 45];
      L     DBD [AR2,P#36.0];
      LAR1;
      CDB;
      L     D [AR1,P#44.0];
      CDB;
      OPN   DI [LW 26];
      T     DID [AR2,P#86.0];
      L     DBW [AR2,P#34.0];
      T     LW 47;
      OPN   DI [LW 47];
      L     DBD [AR2,P#36.0];
      LAR1;
      CDB;
      L     D [AR1,P#48.0];
      CDB;
      OPN   DI [LW 26];
      T     DID [AR2,P#90.0];
      L     L#1065353216;
      T     DID [AR2,P#94.0];
      L     L#0;
      T     DID [AR2,P#98.0];
      L     L#1065353216;
      T     DID [AR2,P#102.0];
      L     L#0;
      T     DID [AR2,P#106.0];
      L     L#0;
      T     DID [AR2,P#110.0];
      L     L#0;
      T     DID [AR2,P#114.0];
      +AR2  P#46.0;
      UC    "CONT_C";
      LAR2  LD 22;
      L     DID [AR2,P#118.0];
      T     LD 8;
      CDB;
      BLD   15;
NETWORK
TITLE =
      BLD   18;
      T     LD 22;
      TAK;
      T     LD 26;
      L     DIW [AR2,P#34.0];
      T     LW 30;
      OPN   DB [LW 30];
      L     DID [AR2,P#36.0];
      LAR1;
      L     LD 26;
      L     LD 22;
      A      [AR1,P#61.3];
      JC    M044;
      BLD   18;
      T     LD 22;
      TAK;
      T     LD 26;
      L     DIW [AR2,P#34.0];
      T     LW 30;
      OPN   DB [LW 30];
      L     DID [AR2,P#36.0];
      LAR1;
      L     LD 26;
      L     LD 22;
      A      [AR1,P#61.0];
      JC    M045;
      L     LD 8;
      JU    M046;
M044: L     DID [AR2,P#18.0];
      JU    M046;
M045: BLD   18;
      T     LD 22;
      TAK;
      T     LD 26;
      L     DIW [AR2,P#34.0];
      T     LW 30;
      OPN   DB [LW 30];
      L     DID [AR2,P#36.0];
      LAR1;
      L     LD 26;
      L     LD 22;
      L     D [AR1,P#16.0];
M046: BLD   18;
      T     LD 22;
      TAK;
      T     LD 26;
      L     DIW [AR2,P#34.0];
      T     LW 30;
      OPN   DB [LW 30];
      L     DID [AR2,P#36.0];
      LAR1;
      L     LD 26;
      L     LD 22;
      T     D [AR1,P#16.0];
      T     DID [AR2,P#28.0];
NETWORK
TITLE =
      SET;
      R     DIX [AR2,P#16.0];
      R     DIX [AR2,P#10.0];
END_FUNCTION_BLOCK

FUNCTION "BatchControlStarch" : VOID	// FC 10
VERSION : 0.1
BEGIN
// (block stored without names or comments; labels and parameter names are numbered)
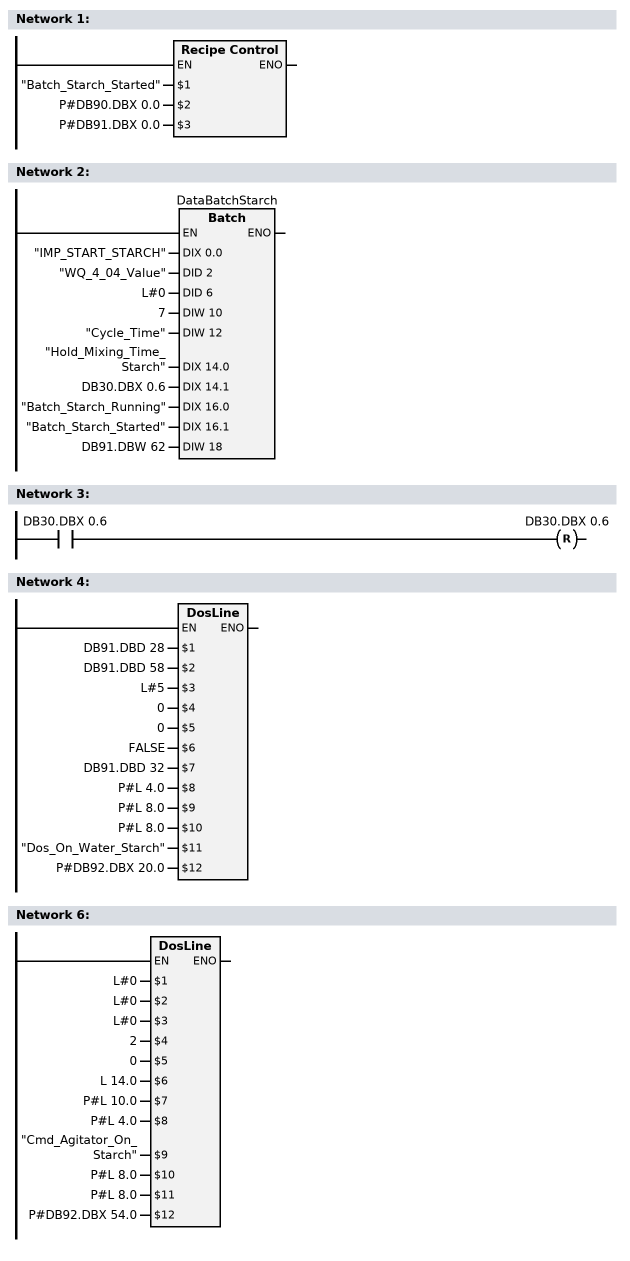
NETWORK
TITLE =
      CALL  "Recipe Control" (
           $1                       := "Batch_Starch_Started",
           $2                       := P#DB90.DBX 0.0,
           $3                       := P#DB91.DBX 0.0);
NETWORK
TITLE =
      CALL  "Batch" , "DataBatchStarch" (
           DIX 0.0                  := "IMP_START_STARCH",
           DID 2                    := "WQ_4_04_Value",
           DID 6                    := L#0,
           DIW 10                   := 7,
           DIW 12                   := "Cycle_Time",
           DIX 14.0                 := "Hold_Mixing_Time_Starch",
           DIX 14.1                 := DB30.DBX 0.6,
           DIX 16.0                 := "Batch_Starch_Running",
           DIX 16.1                 := "Batch_Starch_Started",
           DIW 18                   := DB91.DBW 62);
NETWORK
TITLE =
      A     DB30.DBX 0.6;
      R     DB30.DBX 0.6;
NETWORK
TITLE =
      CALL  "DosLine" (
           $1                       := DB91.DBD 28,
           $2                       := DB91.DBD 58,
           $3                       := L#5,
           $4                       := 0,
           $5                       := 0,
           $6                       := FALSE,
           $7                       := DB91.DBD 32,
           $8                       := P#L 4.0,
           $9                       := P#L 8.0,
           $10                      := P#L 8.0,
           $11                      := "Dos_On_Water_Starch",
           $12                      := P#DB92.DBX 20.0);
NETWORK
TITLE =
      A     "M4_01_RUN";
      L     S5T#20S;
      SD    T 12;
      NOP   0;
      NOP   0;
      NOP   0;
      A     T 12;
      =     L 14.0;
NETWORK
TITLE =
      CALL  "DosLine" (
           $1                       := L#0,
           $2                       := L#0,
           $3                       := L#0,
           $4                       := 2,
           $5                       := 0,
           $6                       := L 14.0,
           $7                       := P#L 10.0,
           $8                       := P#L 4.0,
           $9                       := "Cmd_Agitator_On_Starch",
           $10                      := P#L 8.0,
           $11                      := P#L 8.0,
           $12                      := P#DB92.DBX 54.0);
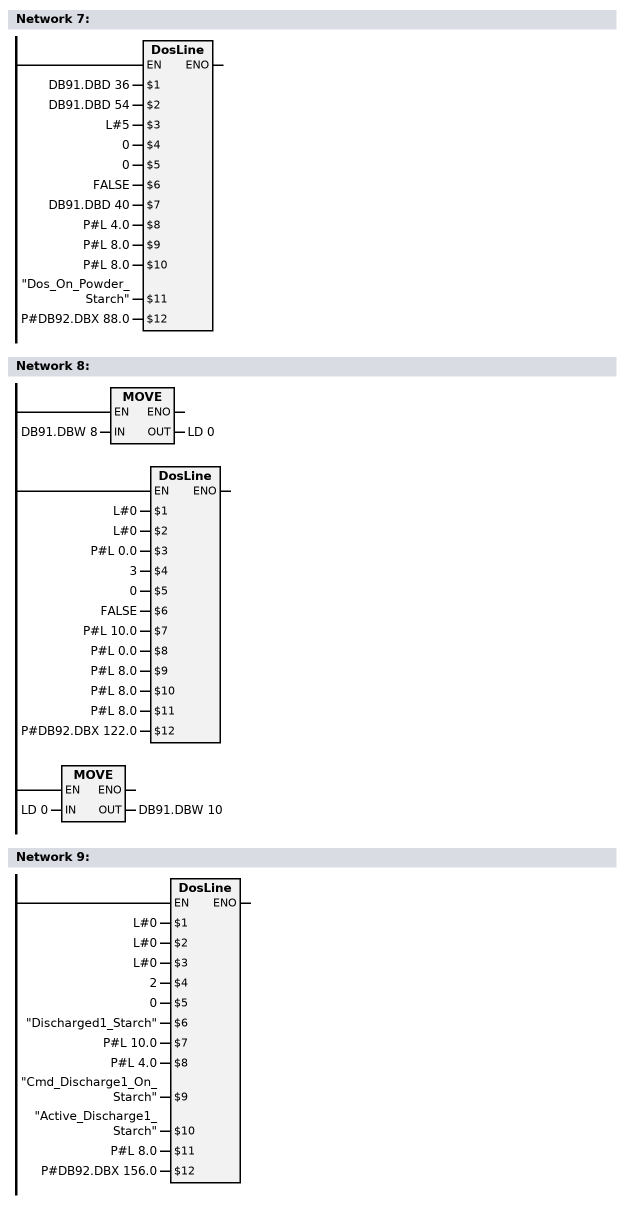
NETWORK
TITLE =
      CALL  "DosLine" (
           $1                       := DB91.DBD 36,
           $2                       := DB91.DBD 54,
           $3                       := L#5,
           $4                       := 0,
           $5                       := 0,
           $6                       := FALSE,
           $7                       := DB91.DBD 40,
           $8                       := P#L 4.0,
           $9                       := P#L 8.0,
           $10                      := P#L 8.0,
           $11                      := "Dos_On_Powder_Starch",
           $12                      := P#DB92.DBX 88.0);
NETWORK
TITLE =
      L     DB91.DBW 8;
      T     LD 0;
      CALL  "DosLine" (
           $1                       := L#0,
           $2                       := L#0,
           $3                       := P#L 0.0,
           $4                       := 3,
           $5                       := 0,
           $6                       := FALSE,
           $7                       := P#L 10.0,
           $8                       := P#L 0.0,
           $9                       := P#L 8.0,
           $10                      := P#L 8.0,
           $11                      := P#L 8.0,
           $12                      := P#DB92.DBX 122.0);
      L     LD 0;
      T     DB91.DBW 10;
NETWORK
TITLE =
      CALL  "DosLine" (
           $1                       := L#0,
           $2                       := L#0,
           $3                       := L#0,
           $4                       := 2,
           $5                       := 0,
           $6                       := "Discharged1_Starch",
           $7                       := P#L 10.0,
           $8                       := P#L 4.0,
           $9                       := "Cmd_Discharge1_On_Starch",
           $10                      := "Active_Discharge1_Starch",
           $11                      := P#L 8.0,
           $12                      := P#DB92.DBX 156.0);
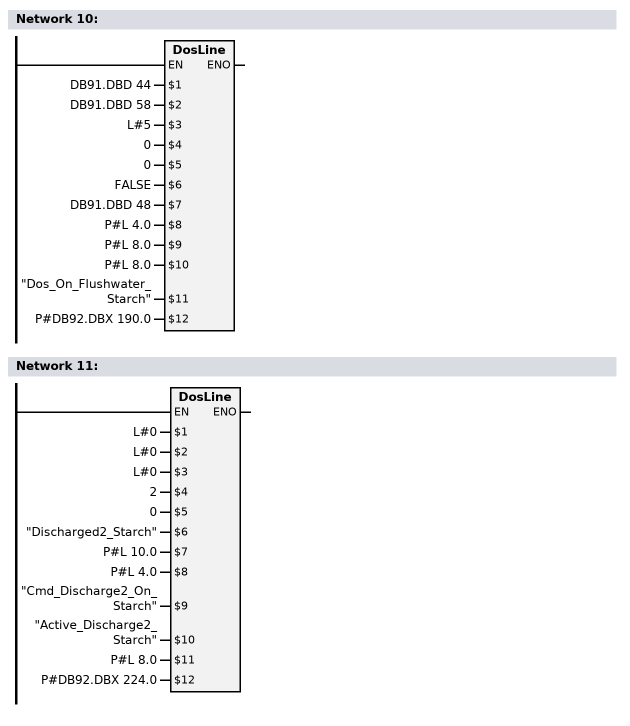
NETWORK
TITLE =
      CALL  "DosLine" (
           $1                       := DB91.DBD 44,
           $2                       := DB91.DBD 58,
           $3                       := L#5,
           $4                       := 0,
           $5                       := 0,
           $6                       := FALSE,
           $7                       := DB91.DBD 48,
           $8                       := P#L 4.0,
           $9                       := P#L 8.0,
           $10                      := P#L 8.0,
           $11                      := "Dos_On_Flushwater_Starch",
           $12                      := P#DB92.DBX 190.0);
NETWORK
TITLE =
      CALL  "DosLine" (
           $1                       := L#0,
           $2                       := L#0,
           $3                       := L#0,
           $4                       := 2,
           $5                       := 0,
           $6                       := "Discharged2_Starch",
           $7                       := P#L 10.0,
           $8                       := P#L 4.0,
           $9                       := "Cmd_Discharge2_On_Starch",
           $10                      := "Active_Discharge2_Starch",
           $11                      := P#L 8.0,
           $12                      := P#DB92.DBX 224.0);
END_FUNCTION

FUNCTION "BatchControlCaCO3" : VOID	// FC 11
VERSION : 0.1
BEGIN
// (block stored without names or comments; labels and parameter names are numbered)
NETWORK
TITLE =
      CALL  "Recipe Control" (
           $1                       := "Batch_CaCO3_Started",
           $2                       := P#DB90.DBX 64.0,
           $3                       := P#DB91.DBX 64.0);
NETWORK
TITLE =
      CALL  "Batch" , "DataBatchCaCO3" (
           DIX 0.0                  := "IMP_START_CaCO3",
           DID 2                    := "WQ_34_04_Value",
           DID 6                    := L#0,
           DIW 10                   := 7,
           DIW 12                   := "Cycle_Time",
           DIX 14.0                 := "Hold_Mixing_Time_CaCO3",
           DIX 14.1                 := DB30.DBX 10.4,
           DIX 16.0                 := "Batch_CaCO3_Running",
           DIX 16.1                 := "Batch_CaCO3_Started",
           DIW 18                   := DB91.DBW 126);
NETWORK
TITLE =
      A     DB30.DBX 10.4;
      R     DB30.DBX 10.4;
NETWORK
TITLE =
      CALL  "DosLine" (
           $1                       := DB91.DBD 92,
           $2                       := DB91.DBD 122,
           $3                       := L#5,
           $4                       := 0,
           $5                       := 0,
           $6                       := FALSE,
           $7                       := DB91.DBD 96,
           $8                       := P#L 4.0,
           $9                       := P#L 8.0,
           $10                      := P#L 8.0,
           $11                      := "Dos_On_Water_CaCO3",
           $12                      := P#DB93.DBX 20.0);
NETWORK
TITLE =
      CALL  "DosLine" (
           $1                       := L#0,
           $2                       := L#0,
           $3                       := L#0,
           $4                       := 2,
           $5                       := 0,
           $6                       := "M34_01_RUN",
           $7                       := P#L 10.0,
           $8                       := P#L 4.0,
           $9                       := "Cmd_Agitator_On_CaCO3",
           $10                      := P#L 8.0,
           $11                      := P#L 8.0,
           $12                      := P#DB93.DBX 54.0);
NETWORK
TITLE =
      CALL  "DosLine" (
           $1                       := DB91.DBD 100,
           $2                       := DB91.DBD 118,
           $3                       := L#1,
           $4                       := 0,
           $5                       := 0,
           $6                       := FALSE,
           $7                       := DB91.DBD 104,
           $8                       := P#L 4.0,
           $9                       := P#L 8.0,
           $10                      := P#L 8.0,
           $11                      := "Dos_On_Powder_CaCO3",
           $12                      := P#DB93.DBX 88.0);
NETWORK
TITLE =
      L     DB91.DBW 72;
      T     LD 0;
      CALL  "DosLine" (
           $1                       := L#0,
           $2                       := L#0,
           $3                       := P#L 0.0,
           $4                       := 3,
           $5                       := 0,
           $6                       := FALSE,
           $7                       := P#L 10.0,
           $8                       := P#L 0.0,
           $9                       := P#L 8.0,
           $10                      := P#L 8.0,
           $11                      := P#L 8.0,
           $12                      := P#DB93.DBX 122.0);
      L     LD 0;
      T     DB91.DBW 74;
NETWORK
TITLE =
      CALL  "DosLine" (
           $1                       := L#0,
           $2                       := L#0,
           $3                       := L#0,
           $4                       := 2,
           $5                       := 0,
           $6                       := "Discharged1_CaCO3",
           $7                       := P#L 10.0,
           $8                       := P#L 4.0,
           $9                       := "Cmd_Discharge1_On_CaCO3",
           $10                      := "Active_Discharge1_CaCO3",
           $11                      := P#L 8.0,
           $12                      := P#DB93.DBX 156.0);
NETWORK
TITLE =
      CALL  "DosLine" (
           $1                       := DB91.DBD 108,
           $2                       := DB91.DBD 122,
           $3                       := L#5,
           $4                       := 0,
           $5                       := 0,
           $6                       := FALSE,
           $7                       := DB91.DBD 112,
           $8                       := P#L 4.0,
           $9                       := P#L 8.0,
           $10                      := P#L 8.0,
           $11                      := "Dos_On_Flushwater_CaCO3",
           $12                      := P#DB93.DBX 190.0);
NETWORK
TITLE =
      CALL  "DosLine" (
           $1                       := L#0,
           $2                       := L#0,
           $3                       := L#0,
           $4                       := 2,
           $5                       := 0,
           $6                       := "Discharged2_CaCO3",
           $7                       := P#L 10.0,
           $8                       := P#L 4.0,
           $9                       := "Cmd_Discharge2_On_CaCO3",
           $10                      := "Active_Discharge2_CaCO3",
           $11                      := P#L 8.0,
           $12                      := P#DB93.DBX 224.0);
END_FUNCTION

